SPLINE
SPL {X  -158.227, Y  +353.814, Z    +0.000, E1   +70.663, E3 +51533.806}
SPL {X  -154.257, Y  +335.055, Z    +0.000, E1   +71.089, E3 +51543.434}
SPL {X  -148.153, Y  +317.104, Z    +0.000, E1   +71.658, E3 +51550.580}
SPL {X  -143.479, Y  +306.716, Z    +0.000, E1   +71.847, E3 +51555.654}
SPL {X  -140.298, Y  +300.601, Z    +0.000, E1   +71.461, E3 +51562.409}
SPL {X  -137.001, Y  +294.872, Z    +0.000, E1   +71.048, E3 +51568.917}
SPL {X  -133.301, Y  +289.026, Z    +0.000, E1   +70.567, E3 +51575.704}
SPL {X  -128.648, Y  +282.387, Z    +0.000, E1   +69.939, E3 +51583.519}
SPL {X  -125.063, Y  +277.720, Z    +0.000, E1   +69.378, E3 +51589.095}
SPL {X  -122.086, Y  +274.099, Z    +0.000, E1   +68.932, E3 +51593.340}
SPL {X   -84.117, Y  +241.407, Z    +0.000, E1   +58.224, E3 +51684.223}
ENDSPLINE

SPLINE
SPL {X  -106.708, Y  +258.294, Z    +0.000, E1   +53.789, E3 +51863.010}
SPL {X  -137.973, Y  +296.505, Z    +0.000, E1   +48.844, E3 +51901.790}
SPL {X  -154.359, Y  +335.426, Z    +0.000, E1   +34.338, E3 +51914.686}
SPL {X  -159.279, Y  +362.429, Z    +0.000, E1   +16.013, E3 +51918.286}
SPL {X  -159.976, Y  +375.387, Z    +0.000, E1    +4.229, E3 +51918.937}
SPL {X  -159.990, Y  +379.485, Z    +0.000, E1    +0.028, E3 +51918.982}
SPL {X  -159.990, Y  +381.270, Z    +0.000, E1    -3.383, E3 +51918.999}
SPL {X  -159.990, Y  +384.811, Z    +0.000, E1   -11.531, E3 +51919.089}
SPL {X  -159.990, Y  +390.180, Z    +0.000, E1   -24.142, E3 +51919.392}
SPL {X  -159.990, Y  +397.074, Z    +0.000, E1   -39.012, E3 +51920.002}
SPL {X  -159.990, Y  +405.152, Z    +0.000, E1   -50.697, E3 +51921.141}
SPL {X  -159.990, Y  +423.293, Z    +0.000, E1   -63.280, E3 +51925.143}
SPL {X  -159.990, Y  +493.649, Z    +0.000, E1   -71.671, E3 +51950.847}
SPL {X  -159.990, Y  +662.531, Z    +0.000, E1   -73.010, E3 +52037.670}
SPL {X  -159.805, Y  +684.185, Z    +0.000, E1   -72.979, E3 +52051.954}
SPL {X  -158.739, Y  +696.464, Z    +0.000, E1   -72.862, E3 +52061.072}
SPL {X  -156.417, Y  +710.124, Z    +0.000, E1   -72.650, E3 +52072.296}
SPL {X  -153.206, Y  +722.596, Z    +0.000, E1   -72.287, E3 +52083.734}
SPL {X  -150.445, Y  +730.933, Z    +0.000, E1   -71.979, E3 +52091.944}
SPL {X  -147.389, Y  +738.737, Z    +0.000, E1   -71.634, E3 +52100.017}
SPL {X  -144.044, Y  +746.129, Z    +0.000, E1   -71.236, E3 +52108.011}
SPL {X  -140.684, Y  +752.689, Z    +0.000, E1   -70.820, E3 +52115.387}
SPL {X  -137.335, Y  +758.572, Z    +0.000, E1   -70.388, E3 +52122.194}
SPL {X  -134.566, Y  +763.037, Z    +0.000, E1   -70.007, E3 +52127.490}
SPL {X  -131.456, Y  +767.693, Z    +0.000, E1   -69.587, E3 +52133.054}
SPL {X  -127.440, Y  +773.226, Z    +0.000, E1   -69.006, E3 +52139.737}
SPL {X  -123.127, Y  +778.659, Z    +0.000, E1   -68.349, E3 +52146.279}
SPL {X   -80.879, Y  +814.541, Z    +0.000, E1   -55.704, E3 +52269.184}
ENDSPLINE

SPLINE
SPL {X  -125.518, Y  +775.707, Z    +0.000, E1   -52.189, E3 +52440.661}
SPL {X  -144.748, Y  +744.653, Z    +0.000, E1   -45.208, E3 +52458.857}
SPL {X  -153.147, Y  +722.791, Z    +0.000, E1   -36.417, E3 +52465.252}
SPL {X  -157.402, Y  +705.160, Z    +0.000, E1   -26.108, E3 +52468.348}
SPL {X  -159.480, Y  +689.270, Z    +0.000, E1   -14.023, E3 +52469.913}
SPL {X  -159.986, Y  +677.650, Z    +0.000, E1    -3.291, E3 +52470.408}
SPL {X  -159.990, Y  +674.500, Z    +0.000, E1    +0.000, E3 +52470.438}
SPL {X  -159.990, Y  +672.716, Z    +0.000, E1    +3.405, E3 +52470.455}
SPL {X  -159.990, Y  +668.521, Z    +0.000, E1   +13.007, E3 +52470.574}
SPL {X  -159.990, Y  +662.839, Z    +0.000, E1   +26.519, E3 +52470.916}
SPL {X  -159.990, Y  +653.836, Z    +0.000, E1   +43.967, E3 +52471.846}
SPL {X  -159.990, Y  +641.022, Z    +0.000, E1   +57.726, E3 +52474.155}
SPL {X  -159.990, Y  +617.987, Z    +0.000, E1   +67.134, E3 +52480.051}
SPL {X  -159.990, Y  +532.407, Z    +0.000, E1   +73.084, E3 +52510.957}
SPL {X  -159.990, Y  +382.957, Z    +0.000, E1   +73.647, E3 +52587.217}
SPL {X  -159.615, Y  +366.548, Z    +0.000, E1   +73.602, E3 +52597.859}
SPL {X  -157.928, Y  +351.899, Z    +0.000, E1   +73.451, E3 +52608.714}
ENDSPLINE

SPLINE
SPL {X  -159.990, Y  +380.170, Z    +0.000, E1   +69.785, E3 +52624.854}
ENDSPLINE

SPLINE
SPL {X  -158.227, Y  +353.814, Z    +0.000, E1   +70.663, E3 +52636.748}
SPL {X  -155.560, Y  +340.111, Z    +0.000, E1   +70.976, E3 +52643.770}
SPL {X  -151.918, Y  +327.322, Z    +0.000, E1   +71.266, E3 +52650.113}
SPL {X  -144.697, Y  +309.238, Z    +0.000, E1   +71.848, E3 +52657.063}
SPL {X  -140.298, Y  +300.601, Z    +0.000, E1   +71.461, E3 +52665.350}
SPL {X  -135.903, Y  +293.078, Z    +0.000, E1   +70.930, E3 +52673.888}
SPL {X  -130.487, Y  +284.926, Z    +0.000, E1   +70.202, E3 +52683.447}
SPL {X  -125.807, Y  +278.659, Z    +0.000, E1   +69.508, E3 +52690.904}
SPL {X  -122.967, Y  +275.148, Z    +0.000, E1   +69.053, E3 +52695.073}
SPL {X  -121.236, Y  +273.103, Z    +0.000, E1   +68.779, E3 +52697.458}
SPL {X   -84.117, Y  +241.407, Z    +0.000, E1   +58.224, E3 +52787.164}
ENDSPLINE

SPLINE
SPL {X  -106.708, Y  +258.294, Z    +0.000, E1   +53.789, E3 +52965.951}
SPL {X  -137.973, Y  +296.505, Z    +0.000, E1   +48.844, E3 +53004.731}
SPL {X  -150.692, Y  +323.752, Z    +0.000, E1   +39.895, E3 +53015.097}
SPL {X  -157.053, Y  +346.986, Z    +0.000, E1   +27.437, E3 +53019.577}
SPL {X  -159.518, Y  +365.226, Z    +0.000, E1   +13.562, E3 +53021.442}
SPL {X  -159.976, Y  +375.387, Z    +0.000, E1    +4.229, E3 +53021.878}
SPL {X  -159.990, Y  +379.485, Z    +0.000, E1    +0.028, E3 +53021.923}
SPL {X  -159.990, Y  +381.270, Z    +0.000, E1    -3.383, E3 +53021.940}
SPL {X  -159.990, Y  +384.811, Z    +0.000, E1   -11.531, E3 +53022.030}
SPL {X  -159.990, Y  +390.180, Z    +0.000, E1   -24.142, E3 +53022.333}
SPL {X  -159.990, Y  +397.074, Z    +0.000, E1   -39.012, E3 +53022.943}
SPL {X  -159.990, Y  +405.152, Z    +0.000, E1   -50.697, E3 +53024.082}
SPL {X  -159.990, Y  +423.293, Z    +0.000, E1   -63.280, E3 +53028.084}
SPL {X  -159.990, Y  +493.649, Z    +0.000, E1   -71.671, E3 +53053.788}
SPL {X  -159.990, Y  +662.531, Z    +0.000, E1   -73.010, E3 +53140.611}
SPL {X  -159.805, Y  +684.185, Z    +0.000, E1   -72.979, E3 +53154.895}
SPL {X  -158.739, Y  +696.464, Z    +0.000, E1   -72.862, E3 +53164.014}
SPL {X  -156.417, Y  +710.124, Z    +0.000, E1   -72.650, E3 +53175.237}
SPL {X  -153.206, Y  +722.596, Z    +0.000, E1   -72.287, E3 +53186.675}
SPL {X  -150.445, Y  +730.933, Z    +0.000, E1   -71.979, E3 +53194.885}
SPL {X  -147.389, Y  +738.737, Z    +0.000, E1   -71.634, E3 +53202.958}
SPL {X  -144.044, Y  +746.129, Z    +0.000, E1   -71.236, E3 +53210.952}
SPL {X  -140.684, Y  +752.689, Z    +0.000, E1   -70.820, E3 +53218.328}
SPL {X  -137.335, Y  +758.572, Z    +0.000, E1   -70.388, E3 +53225.135}
SPL {X  -133.651, Y  +764.444, Z    +0.000, E1   -69.897, E3 +53232.087}
SPL {X  -129.492, Y  +770.461, Z    +0.000, E1   -69.311, E3 +53239.327}
SPL {X  -125.168, Y  +776.148, Z    +0.000, E1   -68.666, E3 +53246.204}
SPL {X  -122.036, Y  +779.960, Z    +0.000, E1   -68.144, E3 +53250.807}
SPL {X   -80.879, Y  +814.541, Z    +0.000, E1   -55.704, E3 +53372.125}
ENDSPLINE

SPLINE
SPL {X  -125.518, Y  +775.707, Z    +0.000, E1   -52.189, E3 +53543.602}
SPL {X  -144.748, Y  +744.653, Z    +0.000, E1   -45.208, E3 +53561.798}
SPL {X  -153.147, Y  +722.791, Z    +0.000, E1   -36.417, E3 +53568.194}
SPL {X  -158.456, Y  +698.602, Z    +0.000, E1   -21.523, E3 +53572.040}
SPL {X  -159.738, Y  +685.469, Z    +0.000, E1   -10.595, E3 +53573.094}
SPL {X  -159.986, Y  +677.650, Z    +0.000, E1    -3.291, E3 +53573.349}
SPL {X  -159.990, Y  +674.500, Z    +0.000, E1    +0.000, E3 +53573.379}
SPL {X  -159.990, Y  +672.716, Z    +0.000, E1    +3.405, E3 +53573.396}
SPL {X  -159.990, Y  +668.521, Z    +0.000, E1   +13.007, E3 +53573.515}
SPL {X  -159.990, Y  +662.839, Z    +0.000, E1   +26.519, E3 +53573.857}
SPL {X  -159.990, Y  +653.836, Z    +0.000, E1   +43.967, E3 +53574.787}
SPL {X  -159.990, Y  +641.022, Z    +0.000, E1   +57.726, E3 +53577.096}
SPL {X  -159.990, Y  +617.987, Z    +0.000, E1   +67.134, E3 +53582.992}
SPL {X  -159.990, Y  +532.407, Z    +0.000, E1   +73.084, E3 +53613.899}
SPL {X  -159.990, Y  +382.957, Z    +0.000, E1   +73.647, E3 +53690.158}
SPL {X  -159.615, Y  +366.548, Z    +0.000, E1   +73.602, E3 +53700.801}
SPL {X  -157.928, Y  +351.899, Z    +0.000, E1   +73.451, E3 +53711.655}
ENDSPLINE

SPLINE
SPL {X  -159.990, Y  +380.170, Z    +0.000, E1   +69.785, E3 +53727.795}
ENDSPLINE

SPLINE
SPL {X  -158.227, Y  +353.814, Z    +0.000, E1   +70.663, E3 +53739.689}
SPL {X  -155.560, Y  +340.111, Z    +0.000, E1   +70.976, E3 +53746.711}
SPL {X  -151.918, Y  +327.322, Z    +0.000, E1   +71.266, E3 +53753.054}
SPL {X  -144.697, Y  +309.238, Z    +0.000, E1   +71.848, E3 +53760.004}
SPL {X  -140.298, Y  +300.601, Z    +0.000, E1   +71.461, E3 +53768.292}
SPL {X  -135.903, Y  +293.078, Z    +0.000, E1   +70.930, E3 +53776.829}
SPL {X  -132.382, Y  +287.656, Z    +0.000, E1   +70.425, E3 +53783.221}
SPL {X  -128.648, Y  +282.387, Z    +0.000, E1   +69.939, E3 +53789.402}
SPL {X  -125.063, Y  +277.720, Z    +0.000, E1   +69.378, E3 +53794.977}
SPL {X  -122.086, Y  +274.099, Z    +0.000, E1   +68.932, E3 +53799.223}
SPL {X   -84.117, Y  +241.407, Z    +0.000, E1   +58.224, E3 +53890.105}
ENDSPLINE

SPLINE
SPL {X  -116.986, Y  +268.362, Z    +0.000, E1   +53.233, E3 +54084.021}
SPL {X  -146.319, Y  +312.789, Z    +0.000, E1   +44.152, E3 +54114.487}
SPL {X  -155.980, Y  +341.904, Z    +0.000, E1   +30.583, E3 +54121.782}
SPL {X  -159.279, Y  +362.429, Z    +0.000, E1   +16.013, E3 +54124.168}
SPL {X  -159.976, Y  +375.387, Z    +0.000, E1    +4.229, E3 +54124.819}
SPL {X  -159.990, Y  +379.485, Z    +0.000, E1    +0.028, E3 +54124.864}
SPL {X  -159.990, Y  +381.270, Z    +0.000, E1    -3.383, E3 +54124.881}
SPL {X  -159.990, Y  +386.246, Z    +0.000, E1   -14.704, E3 +54125.039}
SPL {X  -159.990, Y  +394.075, Z    +0.000, E1   -32.836, E3 +54125.599}
SPL {X  -159.990, Y  +405.152, Z    +0.000, E1   -50.697, E3 +54127.024}
SPL {X  -159.990, Y  +423.293, Z    +0.000, E1   -63.280, E3 +54131.025}
SPL {X  -159.990, Y  +493.649, Z    +0.000, E1   -71.671, E3 +54156.729}
SPL {X  -159.990, Y  +662.531, Z    +0.000, E1   -73.010, E3 +54243.552}
SPL {X  -159.805, Y  +684.185, Z    +0.000, E1   -72.979, E3 +54257.836}
SPL {X  -158.295, Y  +699.729, Z    +0.000, E1   -72.830, E3 +54269.506}
SPL {X  -155.857, Y  +712.630, Z    +0.000, E1   -72.572, E3 +54280.435}
SPL {X  -153.206, Y  +722.596, Z    +0.000, E1   -72.287, E3 +54289.616}
SPL {X  -150.445, Y  +730.933, Z    +0.000, E1   -71.979, E3 +54297.827}
SPL {X  -147.389, Y  +738.737, Z    +0.000, E1   -71.634, E3 +54305.899}
SPL {X  -144.044, Y  +746.129, Z    +0.000, E1   -71.236, E3 +54313.894}
SPL {X  -140.684, Y  +752.689, Z    +0.000, E1   -70.820, E3 +54321.269}
SPL {X  -137.335, Y  +758.572, Z    +0.000, E1   -70.388, E3 +54328.076}
SPL {X  -133.651, Y  +764.444, Z    +0.000, E1   -69.897, E3 +54335.028}
SPL {X  -129.492, Y  +770.461, Z    +0.000, E1   -69.311, E3 +54342.269}
SPL {X  -125.168, Y  +776.148, Z    +0.000, E1   -68.666, E3 +54349.145}
SPL {X  -122.036, Y  +779.960, Z    +0.000, E1   -68.144, E3 +54353.748}
SPL {X   -80.879, Y  +814.541, Z    +0.000, E1   -55.704, E3 +54475.066}
ENDSPLINE

SPLINE
SPL {X  -125.518, Y  +775.707, Z    +0.000, E1   -52.189, E3 +54646.543}
SPL {X  -144.748, Y  +744.653, Z    +0.000, E1   -45.208, E3 +54664.739}
SPL {X  -153.147, Y  +722.791, Z    +0.000, E1   -36.417, E3 +54671.135}
SPL {X  -157.402, Y  +705.160, Z    +0.000, E1   -26.108, E3 +54674.230}
SPL {X  -159.480, Y  +689.270, Z    +0.000, E1   -14.023, E3 +54675.796}
SPL {X  -159.986, Y  +677.650, Z    +0.000, E1    -3.291, E3 +54676.290}
SPL {X  -159.990, Y  +674.500, Z    +0.000, E1    +0.000, E3 +54676.320}
SPL {X  -159.990, Y  +672.716, Z    +0.000, E1    +3.405, E3 +54676.337}
SPL {X  -159.990, Y  +668.521, Z    +0.000, E1   +13.007, E3 +54676.456}
SPL {X  -159.990, Y  +664.286, Z    +0.000, E1   +23.338, E3 +54676.688}
SPL {X  -159.990, Y  +658.431, Z    +0.000, E1   +35.998, E3 +54677.182}
SPL {X  -159.990, Y  +650.524, Z    +0.000, E1   +48.779, E3 +54678.171}
SPL {X  -159.990, Y  +641.022, Z    +0.000, E1   +57.726, E3 +54680.038}
SPL {X  -159.990, Y  +617.987, Z    +0.000, E1   +67.134, E3 +54685.933}
SPL {X  -159.990, Y  +532.407, Z    +0.000, E1   +73.084, E3 +54716.840}
SPL {X  -159.990, Y  +390.607, Z    +0.000, E1   +73.632, E3 +54788.376}
SPL {X  -159.886, Y  +371.742, Z    +0.000, E1   +73.650, E3 +54800.163}
SPL {X  -157.928, Y  +351.899, Z    +0.000, E1   +73.451, E3 +54814.596}
ENDSPLINE

SPLINE
SPL {X  -159.990, Y  +380.170, Z    +0.000, E1   +69.785, E3 +54830.736}
ENDSPLINE

SPLINE
SPL {X  -158.227, Y  +353.814, Z    +0.000, E1   +70.663, E3 +54842.630}
SPL {X  -154.257, Y  +335.055, Z    +0.000, E1   +71.089, E3 +54852.258}
SPL {X  -148.153, Y  +317.104, Z    +0.000, E1   +71.658, E3 +54859.404}
SPL {X  -143.479, Y  +306.716, Z    +0.000, E1   +71.847, E3 +54864.477}
SPL {X  -140.298, Y  +300.601, Z    +0.000, E1   +71.461, E3 +54871.233}
SPL {X  -137.001, Y  +294.872, Z    +0.000, E1   +71.048, E3 +54877.741}
SPL {X  -133.301, Y  +289.026, Z    +0.000, E1   +70.567, E3 +54884.527}
SPL {X  -129.603, Y  +283.692, Z    +0.000, E1   +70.051, E3 +54890.827}
SPL {X  -125.807, Y  +278.659, Z    +0.000, E1   +69.508, E3 +54896.786}
SPL {X  -122.086, Y  +274.099, Z    +0.000, E1   +68.932, E3 +54902.164}
SPL {X   -84.117, Y  +241.407, Z    +0.000, E1   +58.224, E3 +54993.046}
ENDSPLINE

SPLINE
SPL {X  -116.986, Y  +268.362, Z    +0.000, E1   +53.233, E3 +55186.962}
SPL {X  -146.319, Y  +312.789, Z    +0.000, E1   +44.152, E3 +55217.428}
SPL {X  -157.053, Y  +346.986, Z    +0.000, E1   +27.437, E3 +55225.459}
SPL {X  -159.518, Y  +365.226, Z    +0.000, E1   +13.562, E3 +55227.325}
SPL {X  -159.976, Y  +375.387, Z    +0.000, E1    +4.229, E3 +55227.760}
SPL {X  -159.990, Y  +379.485, Z    +0.000, E1    +0.028, E3 +55227.805}
SPL {X  -159.990, Y  +381.270, Z    +0.000, E1    -3.383, E3 +55227.822}
SPL {X  -159.990, Y  +386.246, Z    +0.000, E1   -14.704, E3 +55227.980}
SPL {X  -159.990, Y  +394.075, Z    +0.000, E1   -32.836, E3 +55228.541}
SPL {X  -159.990, Y  +405.152, Z    +0.000, E1   -50.697, E3 +55229.965}
SPL {X  -159.990, Y  +423.293, Z    +0.000, E1   -63.280, E3 +55233.966}
SPL {X  -159.990, Y  +493.649, Z    +0.000, E1   -71.671, E3 +55259.670}
SPL {X  -159.990, Y  +662.531, Z    +0.000, E1   -73.010, E3 +55346.493}
SPL {X  -159.805, Y  +684.185, Z    +0.000, E1   -72.979, E3 +55360.777}
SPL {X  -158.295, Y  +699.729, Z    +0.000, E1   -72.830, E3 +55372.447}
SPL {X  -155.857, Y  +712.630, Z    +0.000, E1   -72.572, E3 +55383.376}
SPL {X  -153.206, Y  +722.596, Z    +0.000, E1   -72.287, E3 +55392.557}
SPL {X  -150.445, Y  +730.933, Z    +0.000, E1   -71.979, E3 +55400.768}
SPL {X  -147.389, Y  +738.737, Z    +0.000, E1   -71.634, E3 +55408.840}
SPL {X  -144.044, Y  +746.129, Z    +0.000, E1   -71.236, E3 +55416.835}
SPL {X  -140.684, Y  +752.689, Z    +0.000, E1   -70.820, E3 +55424.210}
SPL {X  -136.099, Y  +760.606, Z    +0.000, E1   -70.253, E3 +55433.366}
SPL {X  -131.456, Y  +767.693, Z    +0.000, E1   -69.587, E3 +55441.877}
SPL {X  -127.440, Y  +773.226, Z    +0.000, E1   -69.006, E3 +55448.561}
SPL {X  -123.127, Y  +778.659, Z    +0.000, E1   -68.349, E3 +55455.103}
SPL {X   -80.879, Y  +814.541, Z    +0.000, E1   -55.704, E3 +55578.007}
ENDSPLINE

SPLINE
SPL {X  -125.518, Y  +775.707, Z    +0.000, E1   -52.189, E3 +55749.484}
SPL {X  -150.797, Y  +729.951, Z    +0.000, E1   -39.777, E3 +55772.219}
SPL {X  -157.402, Y  +705.160, Z    +0.000, E1   -26.108, E3 +55777.171}
SPL {X  -159.480, Y  +689.270, Z    +0.000, E1   -14.023, E3 +55778.737}
SPL {X  -159.986, Y  +677.650, Z    +0.000, E1    -3.291, E3 +55779.231}
SPL {X  -159.990, Y  +674.500, Z    +0.000, E1    +0.000, E3 +55779.262}
SPL {X  -159.990, Y  +672.716, Z    +0.000, E1    +3.405, E3 +55779.278}
SPL {X  -159.990, Y  +668.521, Z    +0.000, E1   +13.007, E3 +55779.397}
SPL {X  -159.990, Y  +662.839, Z    +0.000, E1   +26.519, E3 +55779.740}
SPL {X  -159.990, Y  +653.836, Z    +0.000, E1   +43.967, E3 +55780.670}
SPL {X  -159.990, Y  +641.022, Z    +0.000, E1   +57.726, E3 +55782.979}
SPL {X  -159.990, Y  +617.987, Z    +0.000, E1   +67.134, E3 +55788.874}
SPL {X  -159.990, Y  +532.407, Z    +0.000, E1   +73.084, E3 +55819.781}
SPL {X  -159.990, Y  +390.607, Z    +0.000, E1   +73.632, E3 +55891.317}
SPL {X  -159.886, Y  +371.742, Z    +0.000, E1   +73.650, E3 +55903.104}
SPL {X  -157.928, Y  +351.899, Z    +0.000, E1   +73.451, E3 +55917.537}
ENDSPLINE

SPLINE
SPL {X  -159.990, Y  +380.170, Z    +0.000, E1   +69.785, E3 +55933.678}
ENDSPLINE

SPLINE
SPL {X  -158.227, Y  +353.814, Z    +0.000, E1   +70.663, E3 +55945.571}
SPL {X  -155.560, Y  +340.111, Z    +0.000, E1   +70.976, E3 +55952.593}
SPL {X  -151.918, Y  +327.322, Z    +0.000, E1   +71.266, E3 +55958.937}
SPL {X  -144.697, Y  +309.238, Z    +0.000, E1   +71.848, E3 +55965.886}
SPL {X  -140.298, Y  +300.601, Z    +0.000, E1   +71.461, E3 +55974.174}
SPL {X  -135.903, Y  +293.078, Z    +0.000, E1   +70.930, E3 +55982.712}
SPL {X  -130.487, Y  +284.926, Z    +0.000, E1   +70.202, E3 +55992.271}
SPL {X  -125.807, Y  +278.659, Z    +0.000, E1   +69.508, E3 +55999.727}
SPL {X  -122.967, Y  +275.148, Z    +0.000, E1   +69.053, E3 +56003.896}
SPL {X  -121.236, Y  +273.103, Z    +0.000, E1   +68.779, E3 +56006.282}
SPL {X   -84.117, Y  +241.407, Z    +0.000, E1   +58.224, E3 +56095.988}
ENDSPLINE

SPLINE
SPL {X  -116.986, Y  +268.362, Z    +0.000, E1   +53.233, E3 +56289.903}
SPL {X  -146.319, Y  +312.789, Z    +0.000, E1   +44.152, E3 +56320.369}
SPL {X  -157.053, Y  +346.986, Z    +0.000, E1   +27.437, E3 +56328.400}
SPL {X  -159.518, Y  +365.226, Z    +0.000, E1   +13.562, E3 +56330.266}
SPL {X  -159.976, Y  +375.387, Z    +0.000, E1    +4.229, E3 +56330.701}
SPL {X  -159.990, Y  +379.485, Z    +0.000, E1    +0.028, E3 +56330.746}
SPL {X  -159.990, Y  +381.270, Z    +0.000, E1    -3.383, E3 +56330.764}
SPL {X  -159.990, Y  +386.246, Z    +0.000, E1   -14.704, E3 +56330.921}
SPL {X  -159.990, Y  +394.075, Z    +0.000, E1   -32.836, E3 +56331.482}
SPL {X  -159.990, Y  +405.152, Z    +0.000, E1   -50.697, E3 +56332.906}
SPL {X  -159.990, Y  +423.293, Z    +0.000, E1   -63.280, E3 +56336.907}
SPL {X  -159.990, Y  +493.649, Z    +0.000, E1   -71.671, E3 +56362.611}
SPL {X  -159.990, Y  +662.531, Z    +0.000, E1   -73.010, E3 +56449.434}
SPL {X  -159.805, Y  +684.185, Z    +0.000, E1   -72.979, E3 +56463.718}
SPL {X  -158.295, Y  +699.729, Z    +0.000, E1   -72.830, E3 +56475.389}
SPL {X  -155.857, Y  +712.630, Z    +0.000, E1   -72.572, E3 +56486.318}
SPL {X  -153.206, Y  +722.596, Z    +0.000, E1   -72.287, E3 +56495.499}
SPL {X  -150.445, Y  +730.933, Z    +0.000, E1   -71.979, E3 +56503.709}
SPL {X  -147.389, Y  +738.737, Z    +0.000, E1   -71.634, E3 +56511.782}
SPL {X  -144.044, Y  +746.129, Z    +0.000, E1   -71.236, E3 +56519.776}
SPL {X  -140.684, Y  +752.689, Z    +0.000, E1   -70.820, E3 +56527.151}
SPL {X  -136.099, Y  +760.606, Z    +0.000, E1   -70.253, E3 +56536.307}
SPL {X  -131.456, Y  +767.693, Z    +0.000, E1   -69.587, E3 +56544.818}
SPL {X  -127.440, Y  +773.226, Z    +0.000, E1   -69.006, E3 +56551.502}
SPL {X  -123.127, Y  +778.659, Z    +0.000, E1   -68.349, E3 +56558.044}
SPL {X   -80.879, Y  +814.541, Z    +0.000, E1   -55.704, E3 +56680.948}
ENDSPLINE

SPLINE
SPL {X  -125.518, Y  +775.707, Z    +0.000, E1   -52.189, E3 +56852.426}
SPL {X  -150.797, Y  +729.951, Z    +0.000, E1   -39.777, E3 +56875.161}
SPL {X  -158.456, Y  +698.602, Z    +0.000, E1   -21.523, E3 +56880.863}
SPL {X  -159.738, Y  +685.469, Z    +0.000, E1   -10.595, E3 +56881.918}
SPL {X  -159.986, Y  +677.650, Z    +0.000, E1    -3.291, E3 +56882.172}
SPL {X  -159.990, Y  +674.500, Z    +0.000, E1    +0.000, E3 +56882.203}
SPL {X  -159.990, Y  +672.716, Z    +0.000, E1    +3.405, E3 +56882.219}
SPL {X  -159.990, Y  +668.521, Z    +0.000, E1   +13.007, E3 +56882.338}
SPL {X  -159.990, Y  +662.839, Z    +0.000, E1   +26.519, E3 +56882.681}
SPL {X  -159.990, Y  +653.836, Z    +0.000, E1   +43.967, E3 +56883.611}
SPL {X  -159.990, Y  +641.022, Z    +0.000, E1   +57.726, E3 +56885.920}
SPL {X  -159.990, Y  +617.987, Z    +0.000, E1   +67.134, E3 +56891.815}
SPL {X  -159.990, Y  +532.407, Z    +0.000, E1   +73.084, E3 +56922.722}
SPL {X  -159.990, Y  +382.957, Z    +0.000, E1   +73.647, E3 +56998.982}
SPL {X  -159.615, Y  +366.548, Z    +0.000, E1   +73.602, E3 +57009.624}
SPL {X  -157.928, Y  +351.899, Z    +0.000, E1   +73.451, E3 +57020.479}
ENDSPLINE

SPLINE
SPL {X  -159.990, Y  +380.170, Z    +0.000, E1   +69.785, E3 +57036.619}
ENDSPLINE

SPLINE
SPL {X  -158.227, Y  +353.814, Z    +0.000, E1   +70.663, E3 +57048.512}
SPL {X  -154.257, Y  +335.055, Z    +0.000, E1   +71.089, E3 +57058.140}
SPL {X  -148.153, Y  +317.104, Z    +0.000, E1   +71.658, E3 +57065.286}
SPL {X  -143.479, Y  +306.716, Z    +0.000, E1   +71.847, E3 +57070.359}
SPL {X  -140.298, Y  +300.601, Z    +0.000, E1   +71.461, E3 +57077.115}
SPL {X  -137.001, Y  +294.872, Z    +0.000, E1   +71.048, E3 +57083.623}
SPL {X  -133.301, Y  +289.026, Z    +0.000, E1   +70.567, E3 +57090.410}
SPL {X  -128.648, Y  +282.387, Z    +0.000, E1   +69.939, E3 +57098.225}
SPL {X  -125.063, Y  +277.720, Z    +0.000, E1   +69.378, E3 +57103.801}
SPL {X  -122.086, Y  +274.099, Z    +0.000, E1   +68.932, E3 +57108.046}
SPL {X   -84.117, Y  +241.407, Z    +0.000, E1   +58.224, E3 +57198.929}
ENDSPLINE

SPLINE
SPL {X  -106.708, Y  +258.294, Z    +0.000, E1   +53.789, E3 +57377.716}
SPL {X  -137.973, Y  +296.505, Z    +0.000, E1   +48.844, E3 +57416.496}
SPL {X  -154.359, Y  +335.426, Z    +0.000, E1   +34.338, E3 +57429.392}
SPL {X  -159.279, Y  +362.429, Z    +0.000, E1   +16.013, E3 +57432.992}
SPL {X  -159.976, Y  +375.387, Z    +0.000, E1    +4.229, E3 +57433.643}
SPL {X  -159.990, Y  +379.485, Z    +0.000, E1    +0.028, E3 +57433.688}
SPL {X  -159.990, Y  +381.270, Z    +0.000, E1    -3.383, E3 +57433.705}
SPL {X  -159.990, Y  +386.246, Z    +0.000, E1   -14.704, E3 +57433.862}
SPL {X  -159.990, Y  +394.075, Z    +0.000, E1   -32.836, E3 +57434.423}
SPL {X  -159.990, Y  +405.152, Z    +0.000, E1   -50.697, E3 +57435.847}
SPL {X  -159.990, Y  +423.293, Z    +0.000, E1   -63.280, E3 +57439.849}
SPL {X  -159.990, Y  +493.649, Z    +0.000, E1   -71.671, E3 +57465.552}
SPL {X  -159.990, Y  +662.531, Z    +0.000, E1   -73.010, E3 +57552.376}
SPL {X  -159.805, Y  +684.185, Z    +0.000, E1   -72.979, E3 +57566.660}
SPL {X  -158.739, Y  +696.464, Z    +0.000, E1   -72.862, E3 +57575.778}
SPL {X  -156.417, Y  +710.124, Z    +0.000, E1   -72.650, E3 +57587.002}
SPL {X  -153.206, Y  +722.596, Z    +0.000, E1   -72.287, E3 +57598.440}
SPL {X  -150.445, Y  +730.933, Z    +0.000, E1   -71.979, E3 +57606.650}
SPL {X  -147.389, Y  +738.737, Z    +0.000, E1   -71.634, E3 +57614.723}
SPL {X  -144.044, Y  +746.129, Z    +0.000, E1   -71.236, E3 +57622.717}
SPL {X  -140.684, Y  +752.689, Z    +0.000, E1   -70.820, E3 +57630.092}
SPL {X  -136.099, Y  +760.606, Z    +0.000, E1   -70.253, E3 +57639.248}
SPL {X  -131.456, Y  +767.693, Z    +0.000, E1   -69.587, E3 +57647.760}
SPL {X  -127.440, Y  +773.226, Z    +0.000, E1   -69.006, E3 +57654.443}
SPL {X  -123.127, Y  +778.659, Z    +0.000, E1   -68.349, E3 +57660.985}
SPL {X   -80.879, Y  +814.541, Z    +0.000, E1   -55.704, E3 +57783.889}
ENDSPLINE

SPLINE
SPL {X  -125.518, Y  +775.707, Z    +0.000, E1   -52.189, E3 +57955.367}
SPL {X  -144.748, Y  +744.653, Z    +0.000, E1   -45.208, E3 +57973.563}
SPL {X  -153.147, Y  +722.791, Z    +0.000, E1   -36.417, E3 +57979.958}
SPL {X  -158.456, Y  +698.602, Z    +0.000, E1   -21.523, E3 +57983.804}
SPL {X  -159.738, Y  +685.469, Z    +0.000, E1   -10.595, E3 +57984.859}
SPL {X  -159.986, Y  +677.650, Z    +0.000, E1    -3.291, E3 +57985.114}
SPL {X  -159.990, Y  +674.500, Z    +0.000, E1    +0.000, E3 +57985.144}
SPL {X  -159.990, Y  +672.716, Z    +0.000, E1    +3.405, E3 +57985.161}
SPL {X  -159.990, Y  +668.521, Z    +0.000, E1   +13.007, E3 +57985.280}
SPL {X  -159.990, Y  +662.839, Z    +0.000, E1   +26.519, E3 +57985.622}
SPL {X  -159.990, Y  +653.836, Z    +0.000, E1   +43.967, E3 +57986.552}
SPL {X  -159.990, Y  +641.022, Z    +0.000, E1   +57.726, E3 +57988.861}
SPL {X  -159.990, Y  +617.987, Z    +0.000, E1   +67.134, E3 +57994.757}
SPL {X  -159.990, Y  +532.407, Z    +0.000, E1   +73.084, E3 +58025.663}
SPL {X  -159.990, Y  +390.607, Z    +0.000, E1   +73.632, E3 +58097.199}
SPL {X  -159.886, Y  +371.742, Z    +0.000, E1   +73.650, E3 +58108.986}
SPL {X  -157.928, Y  +351.899, Z    +0.000, E1   +73.451, E3 +58123.420}
ENDSPLINE

SPLINE
SPL {X  -159.990, Y  +387.996, Z    +0.000, E1   +69.509, E3 +58135.850}
ENDSPLINE

SPLINE
SPL {X  -159.889, Y  +371.819, Z    +0.000, E1   +70.046, E3 +58143.577}
SPL {X  -158.227, Y  +353.814, Z    +0.000, E1   +70.663, E3 +58151.454}
SPL {X  -154.257, Y  +335.055, Z    +0.000, E1   +71.089, E3 +58161.082}
SPL {X  -148.153, Y  +317.104, Z    +0.000, E1   +71.658, E3 +58168.227}
SPL {X  -143.479, Y  +306.716, Z    +0.000, E1   +71.847, E3 +58173.301}
SPL {X  -140.298, Y  +300.601, Z    +0.000, E1   +71.461, E3 +58180.056}
SPL {X  -135.903, Y  +293.078, Z    +0.000, E1   +70.930, E3 +58188.594}
SPL {X  -130.487, Y  +284.926, Z    +0.000, E1   +70.202, E3 +58198.153}
SPL {X  -125.807, Y  +278.659, Z    +0.000, E1   +69.508, E3 +58205.610}
SPL {X  -122.967, Y  +275.148, Z    +0.000, E1   +69.053, E3 +58209.779}
SPL {X  -121.236, Y  +273.103, Z    +0.000, E1   +68.779, E3 +58212.164}
SPL {X   -84.117, Y  +241.407, Z    +0.000, E1   +58.224, E3 +58301.870}
ENDSPLINE

SPLINE
SPL {X  -116.986, Y  +268.362, Z    +0.000, E1   +53.233, E3 +58495.785}
SPL {X  -146.319, Y  +312.789, Z    +0.000, E1   +44.152, E3 +58526.252}
SPL {X  -157.053, Y  +346.986, Z    +0.000, E1   +27.437, E3 +58534.283}
SPL {X  -159.518, Y  +365.226, Z    +0.000, E1   +13.562, E3 +58536.148}
SPL {X  -159.976, Y  +375.387, Z    +0.000, E1    +4.229, E3 +58536.584}
SPL {X  -159.990, Y  +379.485, Z    +0.000, E1    +0.028, E3 +58536.629}
SPL {X  -159.990, Y  +381.270, Z    +0.000, E1    -3.383, E3 +58536.646}
SPL {X  -159.990, Y  +384.811, Z    +0.000, E1   -11.531, E3 +58536.736}
SPL {X  -159.990, Y  +388.002, Z    +0.000, E1   -19.281, E3 +58536.886}
SPL {X  -159.990, Y  +394.075, Z    +0.000, E1   -32.836, E3 +58537.364}
SPL {X  -159.990, Y  +405.152, Z    +0.000, E1   -50.697, E3 +58538.788}
SPL {X  -159.990, Y  +423.293, Z    +0.000, E1   -63.280, E3 +58542.790}
SPL {X  -159.990, Y  +493.649, Z    +0.000, E1   -71.671, E3 +58568.494}
SPL {X  -159.990, Y  +654.929, Z    +0.000, E1   -72.988, E3 +58650.443}
SPL {X  -159.990, Y  +668.018, Z    +0.000, E1   -72.989, E3 +58658.936}
SPL {X  -159.805, Y  +684.185, Z    +0.000, E1   -72.979, E3 +58669.601}
SPL {X  -158.295, Y  +699.729, Z    +0.000, E1   -72.830, E3 +58681.271}
SPL {X  -155.857, Y  +712.630, Z    +0.000, E1   -72.572, E3 +58692.200}
SPL {X  -153.206, Y  +722.596, Z    +0.000, E1   -72.287, E3 +58701.381}
SPL {X  -150.445, Y  +730.933, Z    +0.000, E1   -71.979, E3 +58709.591}
SPL {X  -147.389, Y  +738.737, Z    +0.000, E1   -71.634, E3 +58717.664}
SPL {X  -144.044, Y  +746.129, Z    +0.000, E1   -71.236, E3 +58725.658}
SPL {X  -140.684, Y  +752.689, Z    +0.000, E1   -70.820, E3 +58733.034}
SPL {X  -136.099, Y  +760.606, Z    +0.000, E1   -70.253, E3 +58742.189}
SPL {X  -131.456, Y  +767.693, Z    +0.000, E1   -69.587, E3 +58750.701}
SPL {X  -128.507, Y  +771.803, Z    +0.000, E1   -69.145, E3 +58755.683}
SPL {X  -125.168, Y  +776.148, Z    +0.000, E1   -68.666, E3 +58760.910}
SPL {X  -122.036, Y  +779.960, Z    +0.000, E1   -68.144, E3 +58765.513}
SPL {X   -80.879, Y  +814.541, Z    +0.000, E1   -55.704, E3 +58886.831}
ENDSPLINE

SPLINE
SPL {X  -125.518, Y  +775.707, Z    +0.000, E1   -52.189, E3 +59058.308}
SPL {X  -144.748, Y  +744.653, Z    +0.000, E1   -45.208, E3 +59076.504}
SPL {X  -153.147, Y  +722.791, Z    +0.000, E1   -36.417, E3 +59082.900}
SPL {X  -158.456, Y  +698.602, Z    +0.000, E1   -21.523, E3 +59086.746}
SPL {X  -159.738, Y  +685.469, Z    +0.000, E1   -10.595, E3 +59087.800}
SPL {X  -159.986, Y  +677.650, Z    +0.000, E1    -3.291, E3 +59088.055}
SPL {X  -159.990, Y  +674.500, Z    +0.000, E1    +0.000, E3 +59088.085}
SPL {X  -159.990, Y  +672.716, Z    +0.000, E1    +3.405, E3 +59088.102}
SPL {X  -159.990, Y  +668.521, Z    +0.000, E1   +13.007, E3 +59088.221}
SPL {X  -159.990, Y  +664.286, Z    +0.000, E1   +23.338, E3 +59088.452}
SPL {X  -159.990, Y  +658.431, Z    +0.000, E1   +35.998, E3 +59088.947}
SPL {X  -159.990, Y  +650.524, Z    +0.000, E1   +48.779, E3 +59089.935}
SPL {X  -159.990, Y  +641.022, Z    +0.000, E1   +57.726, E3 +59091.802}
SPL {X  -159.990, Y  +617.987, Z    +0.000, E1   +67.134, E3 +59097.698}
SPL {X  -159.990, Y  +532.407, Z    +0.000, E1   +73.084, E3 +59128.605}
SPL {X  -159.990, Y  +382.957, Z    +0.000, E1   +73.647, E3 +59204.864}
SPL {X  -159.615, Y  +366.548, Z    +0.000, E1   +73.602, E3 +59215.507}
SPL {X  -157.928, Y  +351.899, Z    +0.000, E1   +73.451, E3 +59226.361}
ENDSPLINE

SPLINE
SPL {X  -159.990, Y  +380.170, Z    +0.000, E1   +69.785, E3 +59242.501}
ENDSPLINE

SPLINE
SPL {X  -158.227, Y  +353.814, Z    +0.000, E1   +70.663, E3 +59254.395}
SPL {X  -155.560, Y  +340.111, Z    +0.000, E1   +70.976, E3 +59261.417}
SPL {X  -151.918, Y  +327.322, Z    +0.000, E1   +71.266, E3 +59267.760}
SPL {X  -144.697, Y  +309.238, Z    +0.000, E1   +71.848, E3 +59274.710}
SPL {X  -140.298, Y  +300.601, Z    +0.000, E1   +71.461, E3 +59282.997}
SPL {X  -137.001, Y  +294.872, Z    +0.000, E1   +71.048, E3 +59289.506}
SPL {X  -133.301, Y  +289.026, Z    +0.000, E1   +70.567, E3 +59296.292}
SPL {X  -128.648, Y  +282.387, Z    +0.000, E1   +69.939, E3 +59304.107}
SPL {X  -125.063, Y  +277.720, Z    +0.000, E1   +69.378, E3 +59309.683}
SPL {X  -122.086, Y  +274.099, Z    +0.000, E1   +68.932, E3 +59313.928}
SPL {X   -84.117, Y  +241.407, Z    +0.000, E1   +58.224, E3 +59404.811}
ENDSPLINE

SPLINE
SPL {X  -106.708, Y  +258.294, Z    +0.000, E1   +53.789, E3 +59583.598}
SPL {X  -137.973, Y  +296.505, Z    +0.000, E1   +48.844, E3 +59622.378}
SPL {X  -154.359, Y  +335.426, Z    +0.000, E1   +34.338, E3 +59635.274}
SPL {X  -159.279, Y  +362.429, Z    +0.000, E1   +16.013, E3 +59638.874}
SPL {X  -159.976, Y  +375.387, Z    +0.000, E1    +4.229, E3 +59639.525}
SPL {X  -159.990, Y  +379.485, Z    +0.000, E1    +0.028, E3 +59639.570}
SPL {X  -159.990, Y  +381.270, Z    +0.000, E1    -3.383, E3 +59639.587}
SPL {X  -159.990, Y  +384.811, Z    +0.000, E1   -11.531, E3 +59639.677}
SPL {X  -159.990, Y  +390.180, Z    +0.000, E1   -24.142, E3 +59639.980}
SPL {X  -159.990, Y  +397.074, Z    +0.000, E1   -39.012, E3 +59640.590}
SPL {X  -159.990, Y  +405.152, Z    +0.000, E1   -50.697, E3 +59641.730}
SPL {X  -159.990, Y  +423.293, Z    +0.000, E1   -63.280, E3 +59645.731}
SPL {X  -159.990, Y  +493.649, Z    +0.000, E1   -71.671, E3 +59671.435}
SPL {X  -159.990, Y  +662.531, Z    +0.000, E1   -73.010, E3 +59758.258}
SPL {X  -159.805, Y  +684.185, Z    +0.000, E1   -72.979, E3 +59772.542}
SPL {X  -158.295, Y  +699.729, Z    +0.000, E1   -72.830, E3 +59784.212}
SPL {X  -155.857, Y  +712.630, Z    +0.000, E1   -72.572, E3 +59795.141}
SPL {X  -153.206, Y  +722.596, Z    +0.000, E1   -72.287, E3 +59804.322}
SPL {X  -150.445, Y  +730.933, Z    +0.000, E1   -71.979, E3 +59812.532}
SPL {X  -147.389, Y  +738.737, Z    +0.000, E1   -71.634, E3 +59820.605}
SPL {X  -144.044, Y  +746.129, Z    +0.000, E1   -71.236, E3 +59828.600}
SPL {X  -140.684, Y  +752.689, Z    +0.000, E1   -70.820, E3 +59835.975}
SPL {X  -137.335, Y  +758.572, Z    +0.000, E1   -70.388, E3 +59842.782}
SPL {X  -133.651, Y  +764.444, Z    +0.000, E1   -69.897, E3 +59849.734}
SPL {X  -129.492, Y  +770.461, Z    +0.000, E1   -69.311, E3 +59856.974}
SPL {X  -125.168, Y  +776.148, Z    +0.000, E1   -68.666, E3 +59863.851}
SPL {X  -122.036, Y  +779.960, Z    +0.000, E1   -68.144, E3 +59868.454}
SPL {X   -80.879, Y  +814.541, Z    +0.000, E1   -55.704, E3 +59989.772}
ENDSPLINE

SPLINE
SPL {X  -125.518, Y  +775.707, Z    +0.000, E1   -52.189, E3 +60161.249}
SPL {X  -144.748, Y  +744.653, Z    +0.000, E1   -45.208, E3 +60179.445}
SPL {X  -153.147, Y  +722.791, Z    +0.000, E1   -36.417, E3 +60185.841}
SPL {X  -157.402, Y  +705.160, Z    +0.000, E1   -26.108, E3 +60188.936}
SPL {X  -159.480, Y  +689.270, Z    +0.000, E1   -14.023, E3 +60190.502}
SPL {X  -159.986, Y  +677.650, Z    +0.000, E1    -3.291, E3 +60190.996}
SPL {X  -159.990, Y  +674.500, Z    +0.000, E1    +0.000, E3 +60191.026}
SPL {X  -159.990, Y  +672.716, Z    +0.000, E1    +3.405, E3 +60191.043}
SPL {X  -159.990, Y  +668.521, Z    +0.000, E1   +13.007, E3 +60191.162}
SPL {X  -159.990, Y  +664.286, Z    +0.000, E1   +23.338, E3 +60191.393}
SPL {X  -159.990, Y  +658.431, Z    +0.000, E1   +35.998, E3 +60191.888}
SPL {X  -159.990, Y  +650.524, Z    +0.000, E1   +48.779, E3 +60192.877}
SPL {X  -159.990, Y  +641.022, Z    +0.000, E1   +57.726, E3 +60194.743}
SPL {X  -159.990, Y  +617.987, Z    +0.000, E1   +67.134, E3 +60200.639}
SPL {X  -159.990, Y  +532.407, Z    +0.000, E1   +73.084, E3 +60231.546}
SPL {X  -159.990, Y  +390.607, Z    +0.000, E1   +73.632, E3 +60303.082}
SPL {X  -159.886, Y  +371.742, Z    +0.000, E1   +73.650, E3 +60314.869}
SPL {X  -157.928, Y  +351.899, Z    +0.000, E1   +73.451, E3 +60329.302}
ENDSPLINE

SPLINE
SPL {X  -159.990, Y  +380.170, Z    +0.000, E1   +69.785, E3 +60345.442}
ENDSPLINE

SPLINE
SPL {X  -158.227, Y  +353.814, Z    +0.000, E1   +70.663, E3 +60357.336}
SPL {X  -155.560, Y  +340.111, Z    +0.000, E1   +70.976, E3 +60364.358}
SPL {X  -151.918, Y  +327.322, Z    +0.000, E1   +71.266, E3 +60370.702}
SPL {X  -144.697, Y  +309.238, Z    +0.000, E1   +71.848, E3 +60377.651}
SPL {X  -140.298, Y  +300.601, Z    +0.000, E1   +71.461, E3 +60385.939}
SPL {X  -137.001, Y  +294.872, Z    +0.000, E1   +71.048, E3 +60392.447}
SPL {X  -133.301, Y  +289.026, Z    +0.000, E1   +70.567, E3 +60399.233}
SPL {X  -129.603, Y  +283.692, Z    +0.000, E1   +70.051, E3 +60405.533}
SPL {X  -125.807, Y  +278.659, Z    +0.000, E1   +69.508, E3 +60411.492}
SPL {X  -122.086, Y  +274.099, Z    +0.000, E1   +68.932, E3 +60416.870}
SPL {X   -84.117, Y  +241.407, Z    +0.000, E1   +58.224, E3 +60507.752}
ENDSPLINE

SPLINE
SPL {X  -106.708, Y  +258.294, Z    +0.000, E1   +53.789, E3 +60686.539}
SPL {X  -137.973, Y  +296.505, Z    +0.000, E1   +48.844, E3 +60725.319}
SPL {X  -154.359, Y  +335.426, Z    +0.000, E1   +34.338, E3 +60738.215}
SPL {X  -159.279, Y  +362.429, Z    +0.000, E1   +16.013, E3 +60741.815}
SPL {X  -159.976, Y  +375.387, Z    +0.000, E1    +4.229, E3 +60742.466}
SPL {X  -159.990, Y  +379.485, Z    +0.000, E1    +0.028, E3 +60742.511}
SPL {X  -159.990, Y  +381.270, Z    +0.000, E1    -3.383, E3 +60742.528}
SPL {X  -159.990, Y  +386.246, Z    +0.000, E1   -14.704, E3 +60742.686}
SPL {X  -159.990, Y  +394.075, Z    +0.000, E1   -32.836, E3 +60743.246}
SPL {X  -159.990, Y  +405.152, Z    +0.000, E1   -50.697, E3 +60744.671}
SPL {X  -159.990, Y  +423.293, Z    +0.000, E1   -63.280, E3 +60748.672}
SPL {X  -159.990, Y  +493.649, Z    +0.000, E1   -71.671, E3 +60774.376}
SPL {X  -159.990, Y  +662.531, Z    +0.000, E1   -73.010, E3 +60861.199}
SPL {X  -159.805, Y  +684.185, Z    +0.000, E1   -72.979, E3 +60875.483}
SPL {X  -158.295, Y  +699.729, Z    +0.000, E1   -72.830, E3 +60887.153}
SPL {X  -155.857, Y  +712.630, Z    +0.000, E1   -72.572, E3 +60898.082}
SPL {X  -153.206, Y  +722.596, Z    +0.000, E1   -72.287, E3 +60907.263}
SPL {X  -150.445, Y  +730.933, Z    +0.000, E1   -71.979, E3 +60915.474}
SPL {X  -147.389, Y  +738.737, Z    +0.000, E1   -71.634, E3 +60923.546}
SPL {X  -144.044, Y  +746.129, Z    +0.000, E1   -71.236, E3 +60931.541}
SPL {X  -140.684, Y  +752.689, Z    +0.000, E1   -70.820, E3 +60938.916}
SPL {X  -136.099, Y  +760.606, Z    +0.000, E1   -70.253, E3 +60948.071}
SPL {X  -131.456, Y  +767.693, Z    +0.000, E1   -69.587, E3 +60956.583}
SPL {X  -127.440, Y  +773.226, Z    +0.000, E1   -69.006, E3 +60963.267}
SPL {X  -123.127, Y  +778.659, Z    +0.000, E1   -68.349, E3 +60969.809}
SPL {X   -80.879, Y  +814.541, Z    +0.000, E1   -55.704, E3 +61092.713}
ENDSPLINE

SPLINE
SPL {X  -125.518, Y  +775.707, Z    +0.000, E1   -52.189, E3 +61264.190}
SPL {X  -150.797, Y  +729.951, Z    +0.000, E1   -39.777, E3 +61286.925}
SPL {X  -157.402, Y  +705.160, Z    +0.000, E1   -26.108, E3 +61291.877}
SPL {X  -159.480, Y  +689.270, Z    +0.000, E1   -14.023, E3 +61293.443}
SPL {X  -159.986, Y  +677.650, Z    +0.000, E1    -3.291, E3 +61293.937}
SPL {X  -159.990, Y  +674.500, Z    +0.000, E1    +0.000, E3 +61293.968}
SPL {X  -159.990, Y  +672.716, Z    +0.000, E1    +3.405, E3 +61293.984}
SPL {X  -159.990, Y  +668.521, Z    +0.000, E1   +13.007, E3 +61294.103}
SPL {X  -159.990, Y  +662.839, Z    +0.000, E1   +26.519, E3 +61294.445}
SPL {X  -159.990, Y  +653.836, Z    +0.000, E1   +43.967, E3 +61295.376}
SPL {X  -159.990, Y  +641.022, Z    +0.000, E1   +57.726, E3 +61297.685}
SPL {X  -159.990, Y  +617.987, Z    +0.000, E1   +67.134, E3 +61303.580}
SPL {X  -159.990, Y  +532.407, Z    +0.000, E1   +73.084, E3 +61334.487}
SPL {X  -159.990, Y  +390.607, Z    +0.000, E1   +73.632, E3 +61406.023}
SPL {X  -159.886, Y  +371.742, Z    +0.000, E1   +73.650, E3 +61417.810}
SPL {X  -157.928, Y  +351.899, Z    +0.000, E1   +73.451, E3 +61432.243}
ENDSPLINE

SPLINE
SPL {X  -159.990, Y  +380.170, Z    +0.000, E1   +69.785, E3 +61448.384}
ENDSPLINE

SPLINE
SPL {X  -158.227, Y  +353.814, Z    +0.000, E1   +70.663, E3 +61460.277}
SPL {X  -155.560, Y  +340.111, Z    +0.000, E1   +70.976, E3 +61467.299}
SPL {X  -151.918, Y  +327.322, Z    +0.000, E1   +71.266, E3 +61473.643}
SPL {X  -144.697, Y  +309.238, Z    +0.000, E1   +71.848, E3 +61480.592}
SPL {X  -140.298, Y  +300.601, Z    +0.000, E1   +71.461, E3 +61488.880}
SPL {X  -135.903, Y  +293.078, Z    +0.000, E1   +70.930, E3 +61497.417}
SPL {X  -130.487, Y  +284.926, Z    +0.000, E1   +70.202, E3 +61506.977}
SPL {X  -125.807, Y  +278.659, Z    +0.000, E1   +69.508, E3 +61514.433}
SPL {X  -122.967, Y  +275.148, Z    +0.000, E1   +69.053, E3 +61518.602}
SPL {X  -121.236, Y  +273.103, Z    +0.000, E1   +68.779, E3 +61520.988}
SPL {X   -84.117, Y  +241.407, Z    +0.000, E1   +58.224, E3 +61610.693}
ENDSPLINE

SPLINE
SPL {X  -116.986, Y  +268.362, Z    +0.000, E1   +53.233, E3 +61804.609}
SPL {X  -146.319, Y  +312.789, Z    +0.000, E1   +44.152, E3 +61835.075}
SPL {X  -157.053, Y  +346.986, Z    +0.000, E1   +27.437, E3 +61843.106}
SPL {X  -159.518, Y  +365.226, Z    +0.000, E1   +13.562, E3 +61844.972}
SPL {X  -159.976, Y  +375.387, Z    +0.000, E1    +4.229, E3 +61845.407}
SPL {X  -159.990, Y  +379.485, Z    +0.000, E1    +0.028, E3 +61845.452}
SPL {X  -159.990, Y  +381.270, Z    +0.000, E1    -3.383, E3 +61845.469}
SPL {X  -159.990, Y  +386.246, Z    +0.000, E1   -14.704, E3 +61845.627}
SPL {X  -159.990, Y  +394.075, Z    +0.000, E1   -32.836, E3 +61846.188}
SPL {X  -159.990, Y  +405.152, Z    +0.000, E1   -50.697, E3 +61847.612}
SPL {X  -159.990, Y  +423.293, Z    +0.000, E1   -63.280, E3 +61851.613}
SPL {X  -159.990, Y  +493.649, Z    +0.000, E1   -71.671, E3 +61877.317}
SPL {X  -159.990, Y  +662.531, Z    +0.000, E1   -73.010, E3 +61964.140}
SPL {X  -159.805, Y  +684.185, Z    +0.000, E1   -72.979, E3 +61978.424}
SPL {X  -158.295, Y  +699.729, Z    +0.000, E1   -72.830, E3 +61990.095}
SPL {X  -155.857, Y  +712.630, Z    +0.000, E1   -72.572, E3 +62001.024}
SPL {X  -153.206, Y  +722.596, Z    +0.000, E1   -72.287, E3 +62010.204}
SPL {X  -150.445, Y  +730.933, Z    +0.000, E1   -71.979, E3 +62018.415}
SPL {X  -147.389, Y  +738.737, Z    +0.000, E1   -71.634, E3 +62026.487}
SPL {X  -144.044, Y  +746.129, Z    +0.000, E1   -71.236, E3 +62034.482}
SPL {X  -140.684, Y  +752.689, Z    +0.000, E1   -70.820, E3 +62041.857}
SPL {X  -136.099, Y  +760.606, Z    +0.000, E1   -70.253, E3 +62051.013}
SPL {X  -131.456, Y  +767.693, Z    +0.000, E1   -69.587, E3 +62059.524}
SPL {X  -127.440, Y  +773.226, Z    +0.000, E1   -69.006, E3 +62066.208}
SPL {X  -123.127, Y  +778.659, Z    +0.000, E1   -68.349, E3 +62072.750}
SPL {X   -80.879, Y  +814.541, Z    +0.000, E1   -55.704, E3 +62195.654}
ENDSPLINE

SPLINE
SPL {X  -125.518, Y  +775.707, Z    +0.000, E1   -52.189, E3 +62367.132}
SPL {X  -150.797, Y  +729.951, Z    +0.000, E1   -39.777, E3 +62389.866}
SPL {X  -158.456, Y  +698.602, Z    +0.000, E1   -21.523, E3 +62395.569}
SPL {X  -159.738, Y  +685.469, Z    +0.000, E1   -10.595, E3 +62396.623}
SPL {X  -159.986, Y  +677.650, Z    +0.000, E1    -3.291, E3 +62396.878}
SPL {X  -159.990, Y  +674.500, Z    +0.000, E1    +0.000, E3 +62396.909}
SPL {X  -159.990, Y  +672.716, Z    +0.000, E1    +3.405, E3 +62396.925}
SPL {X  -159.990, Y  +668.521, Z    +0.000, E1   +13.007, E3 +62397.044}
SPL {X  -159.990, Y  +662.839, Z    +0.000, E1   +26.519, E3 +62397.387}
SPL {X  -159.990, Y  +653.836, Z    +0.000, E1   +43.967, E3 +62398.317}
SPL {X  -159.990, Y  +641.022, Z    +0.000, E1   +57.726, E3 +62400.626}
SPL {X  -159.990, Y  +617.987, Z    +0.000, E1   +67.134, E3 +62406.521}
SPL {X  -159.990, Y  +532.407, Z    +0.000, E1   +73.084, E3 +62437.428}
SPL {X  -159.990, Y  +382.957, Z    +0.000, E1   +73.647, E3 +62513.688}
SPL {X  -159.615, Y  +366.548, Z    +0.000, E1   +73.602, E3 +62524.330}
SPL {X  -157.928, Y  +351.899, Z    +0.000, E1   +73.451, E3 +62535.184}
ENDSPLINE

SPLINE
SPL {X  -159.990, Y  +380.170, Z    +0.000, E1   +69.785, E3 +62551.325}
ENDSPLINE

SPLINE
SPL {X  -158.227, Y  +353.814, Z    +0.000, E1   +70.663, E3 +62563.218}
SPL {X  -154.257, Y  +335.055, Z    +0.000, E1   +71.089, E3 +62572.846}
SPL {X  -148.153, Y  +317.104, Z    +0.000, E1   +71.658, E3 +62579.992}
SPL {X  -143.479, Y  +306.716, Z    +0.000, E1   +71.847, E3 +62585.065}
SPL {X  -140.298, Y  +300.601, Z    +0.000, E1   +71.461, E3 +62591.821}
SPL {X  -137.001, Y  +294.872, Z    +0.000, E1   +71.048, E3 +62598.329}
SPL {X  -133.301, Y  +289.026, Z    +0.000, E1   +70.567, E3 +62605.116}
SPL {X  -128.648, Y  +282.387, Z    +0.000, E1   +69.939, E3 +62612.931}
SPL {X  -125.063, Y  +277.720, Z    +0.000, E1   +69.378, E3 +62618.507}
SPL {X  -122.086, Y  +274.099, Z    +0.000, E1   +68.932, E3 +62622.752}
SPL {X   -84.117, Y  +241.407, Z    +0.000, E1   +58.224, E3 +62713.635}
ENDSPLINE

SPLINE
SPL {X  -106.708, Y  +258.294, Z    +0.000, E1   +53.789, E3 +62892.422}
SPL {X  -137.973, Y  +296.505, Z    +0.000, E1   +48.844, E3 +62931.202}
SPL {X  -154.359, Y  +335.426, Z    +0.000, E1   +34.338, E3 +62944.098}
SPL {X  -159.279, Y  +362.429, Z    +0.000, E1   +16.013, E3 +62947.698}
SPL {X  -159.976, Y  +375.387, Z    +0.000, E1    +4.229, E3 +62948.348}
SPL {X  -159.990, Y  +379.485, Z    +0.000, E1    +0.028, E3 +62948.394}
SPL {X  -159.990, Y  +381.270, Z    +0.000, E1    -3.383, E3 +62948.411}
SPL {X  -159.990, Y  +384.811, Z    +0.000, E1   -11.531, E3 +62948.501}
SPL {X  -159.990, Y  +390.180, Z    +0.000, E1   -24.142, E3 +62948.804}
SPL {X  -159.990, Y  +397.074, Z    +0.000, E1   -39.012, E3 +62949.414}
SPL {X  -159.990, Y  +405.152, Z    +0.000, E1   -50.697, E3 +62950.553}
SPL {X  -159.990, Y  +423.293, Z    +0.000, E1   -63.280, E3 +62954.554}
SPL {X  -159.990, Y  +493.649, Z    +0.000, E1   -71.671, E3 +62980.258}
SPL {X  -159.990, Y  +662.531, Z    +0.000, E1   -73.010, E3 +63067.081}
SPL {X  -159.805, Y  +684.185, Z    +0.000, E1   -72.979, E3 +63081.365}
SPL {X  -158.739, Y  +696.464, Z    +0.000, E1   -72.862, E3 +63090.484}
SPL {X  -156.417, Y  +710.124, Z    +0.000, E1   -72.650, E3 +63101.707}
SPL {X  -153.206, Y  +722.596, Z    +0.000, E1   -72.287, E3 +63113.146}
SPL {X  -150.445, Y  +730.933, Z    +0.000, E1   -71.979, E3 +63121.356}
SPL {X  -147.389, Y  +738.737, Z    +0.000, E1   -71.634, E3 +63129.429}
SPL {X  -144.044, Y  +746.129, Z    +0.000, E1   -71.236, E3 +63137.423}
SPL {X  -140.684, Y  +752.689, Z    +0.000, E1   -70.820, E3 +63144.798}
SPL {X  -137.335, Y  +758.572, Z    +0.000, E1   -70.388, E3 +63151.606}
SPL {X  -134.566, Y  +763.037, Z    +0.000, E1   -70.007, E3 +63156.902}
SPL {X  -131.456, Y  +767.693, Z    +0.000, E1   -69.587, E3 +63162.465}
SPL {X  -127.440, Y  +773.226, Z    +0.000, E1   -69.006, E3 +63169.149}
SPL {X  -123.127, Y  +778.659, Z    +0.000, E1   -68.349, E3 +63175.691}
SPL {X   -80.879, Y  +814.541, Z    +0.000, E1   -55.704, E3 +63298.595}
ENDSPLINE

SPLINE
SPL {X  -125.518, Y  +775.707, Z    +0.000, E1   -52.189, E3 +63470.073}
SPL {X  -144.748, Y  +744.653, Z    +0.000, E1   -45.208, E3 +63488.269}
SPL {X  -153.147, Y  +722.791, Z    +0.000, E1   -36.417, E3 +63494.664}
SPL {X  -157.402, Y  +705.160, Z    +0.000, E1   -26.108, E3 +63497.759}
SPL {X  -159.480, Y  +689.270, Z    +0.000, E1   -14.023, E3 +63499.325}
SPL {X  -159.986, Y  +677.650, Z    +0.000, E1    -3.291, E3 +63499.819}
SPL {X  -159.990, Y  +674.500, Z    +0.000, E1    +0.000, E3 +63499.850}
SPL {X  -159.990, Y  +672.716, Z    +0.000, E1    +3.405, E3 +63499.866}
SPL {X  -159.990, Y  +668.521, Z    +0.000, E1   +13.007, E3 +63499.985}
SPL {X  -159.990, Y  +662.839, Z    +0.000, E1   +26.519, E3 +63500.328}
SPL {X  -159.990, Y  +653.836, Z    +0.000, E1   +43.967, E3 +63501.258}
SPL {X  -159.990, Y  +641.022, Z    +0.000, E1   +57.726, E3 +63503.567}
SPL {X  -159.990, Y  +617.987, Z    +0.000, E1   +67.134, E3 +63509.463}
SPL {X  -159.990, Y  +532.407, Z    +0.000, E1   +73.084, E3 +63540.369}
SPL {X  -159.990, Y  +382.957, Z    +0.000, E1   +73.647, E3 +63616.629}
SPL {X  -159.615, Y  +366.548, Z    +0.000, E1   +73.602, E3 +63627.271}
SPL {X  -157.928, Y  +351.899, Z    +0.000, E1   +73.451, E3 +63638.126}
ENDSPLINE

SPLINE
SPL {X  -159.990, Y  +380.170, Z    +0.000, E1   +69.785, E3 +63654.266}
ENDSPLINE

SPLINE
SPL {X  -158.227, Y  +353.814, Z    +0.000, E1   +70.663, E3 +63666.159}
SPL {X  -155.560, Y  +340.111, Z    +0.000, E1   +70.976, E3 +63673.181}
SPL {X  -151.918, Y  +327.322, Z    +0.000, E1   +71.266, E3 +63679.525}
SPL {X  -144.697, Y  +309.238, Z    +0.000, E1   +71.848, E3 +63686.475}
SPL {X  -140.298, Y  +300.601, Z    +0.000, E1   +71.461, E3 +63694.762}
SPL {X  -135.903, Y  +293.078, Z    +0.000, E1   +70.930, E3 +63703.300}
SPL {X  -130.487, Y  +284.926, Z    +0.000, E1   +70.202, E3 +63712.859}
SPL {X  -125.807, Y  +278.659, Z    +0.000, E1   +69.508, E3 +63720.316}
SPL {X  -122.967, Y  +275.148, Z    +0.000, E1   +69.053, E3 +63724.484}
SPL {X  -121.236, Y  +273.103, Z    +0.000, E1   +68.779, E3 +63726.870}
SPL {X   -84.117, Y  +241.407, Z    +0.000, E1   +58.224, E3 +63816.576}
ENDSPLINE

SPLINE
SPL {X  -106.708, Y  +258.294, Z    +0.000, E1   +53.789, E3 +63995.363}
SPL {X  -137.973, Y  +296.505, Z    +0.000, E1   +48.844, E3 +64034.143}
SPL {X  -150.692, Y  +323.752, Z    +0.000, E1   +39.895, E3 +64044.509}
SPL {X  -157.053, Y  +346.986, Z    +0.000, E1   +27.437, E3 +64048.989}
SPL {X  -159.518, Y  +365.226, Z    +0.000, E1   +13.562, E3 +64050.854}
SPL {X  -159.976, Y  +375.387, Z    +0.000, E1    +4.229, E3 +64051.290}
SPL {X  -159.990, Y  +379.485, Z    +0.000, E1    +0.028, E3 +64051.335}
SPL {X  -159.990, Y  +381.270, Z    +0.000, E1    -3.383, E3 +64051.352}
SPL {X  -159.990, Y  +384.811, Z    +0.000, E1   -11.531, E3 +64051.442}
SPL {X  -159.990, Y  +390.180, Z    +0.000, E1   -24.142, E3 +64051.745}
SPL {X  -159.990, Y  +397.074, Z    +0.000, E1   -39.012, E3 +64052.355}
SPL {X  -159.990, Y  +405.152, Z    +0.000, E1   -50.697, E3 +64053.494}
SPL {X  -159.990, Y  +423.293, Z    +0.000, E1   -63.280, E3 +64057.496}
SPL {X  -159.990, Y  +493.649, Z    +0.000, E1   -71.671, E3 +64083.199}
SPL {X  -159.990, Y  +662.531, Z    +0.000, E1   -73.010, E3 +64170.023}
SPL {X  -159.805, Y  +684.185, Z    +0.000, E1   -72.979, E3 +64184.307}
SPL {X  -158.739, Y  +696.464, Z    +0.000, E1   -72.862, E3 +64193.425}
SPL {X  -156.417, Y  +710.124, Z    +0.000, E1   -72.650, E3 +64204.649}
SPL {X  -153.206, Y  +722.596, Z    +0.000, E1   -72.287, E3 +64216.087}
SPL {X  -150.445, Y  +730.933, Z    +0.000, E1   -71.979, E3 +64224.297}
SPL {X  -147.389, Y  +738.737, Z    +0.000, E1   -71.634, E3 +64232.370}
SPL {X  -144.044, Y  +746.129, Z    +0.000, E1   -71.236, E3 +64240.364}
SPL {X  -140.684, Y  +752.689, Z    +0.000, E1   -70.820, E3 +64247.740}
SPL {X  -137.335, Y  +758.572, Z    +0.000, E1   -70.388, E3 +64254.547}
SPL {X  -133.651, Y  +764.444, Z    +0.000, E1   -69.897, E3 +64261.499}
SPL {X  -129.492, Y  +770.461, Z    +0.000, E1   -69.311, E3 +64268.739}
SPL {X  -125.168, Y  +776.148, Z    +0.000, E1   -68.666, E3 +64275.615}
SPL {X  -122.036, Y  +779.960, Z    +0.000, E1   -68.144, E3 +64280.219}
SPL {X   -80.879, Y  +814.541, Z    +0.000, E1   -55.704, E3 +64401.536}
ENDSPLINE

SPLINE
SPL {X  -125.518, Y  +775.707, Z    +0.000, E1   -52.189, E3 +64573.014}
SPL {X  -144.748, Y  +744.653, Z    +0.000, E1   -45.208, E3 +64591.210}
SPL {X  -153.147, Y  +722.791, Z    +0.000, E1   -36.417, E3 +64597.605}
SPL {X  -158.456, Y  +698.602, Z    +0.000, E1   -21.523, E3 +64601.451}
SPL {X  -159.738, Y  +685.469, Z    +0.000, E1   -10.595, E3 +64602.506}
SPL {X  -159.986, Y  +677.650, Z    +0.000, E1    -3.291, E3 +64602.761}
SPL {X  -159.990, Y  +674.500, Z    +0.000, E1    +0.000, E3 +64602.791}
SPL {X  -159.990, Y  +672.716, Z    +0.000, E1    +3.405, E3 +64602.808}
SPL {X  -159.990, Y  +668.521, Z    +0.000, E1   +13.007, E3 +64602.927}
SPL {X  -159.990, Y  +662.839, Z    +0.000, E1   +26.519, E3 +64603.269}
SPL {X  -159.990, Y  +653.836, Z    +0.000, E1   +43.967, E3 +64604.199}
SPL {X  -159.990, Y  +641.022, Z    +0.000, E1   +57.726, E3 +64606.508}
SPL {X  -159.990, Y  +617.987, Z    +0.000, E1   +67.134, E3 +64612.404}
SPL {X  -159.990, Y  +532.407, Z    +0.000, E1   +73.084, E3 +64643.310}
SPL {X  -159.990, Y  +382.957, Z    +0.000, E1   +73.647, E3 +64719.570}
SPL {X  -159.615, Y  +366.548, Z    +0.000, E1   +73.602, E3 +64730.212}
SPL {X  -157.928, Y  +351.899, Z    +0.000, E1   +73.451, E3 +64741.067}
ENDSPLINE

SPLINE
SPL {X  -159.990, Y  +380.170, Z    +0.000, E1   +69.785, E3 +64757.207}
ENDSPLINE

SPLINE
SPL {X  -158.227, Y  +353.814, Z    +0.000, E1   +70.663, E3 +64769.101}
SPL {X  -155.560, Y  +340.111, Z    +0.000, E1   +70.976, E3 +64776.123}
SPL {X  -151.918, Y  +327.322, Z    +0.000, E1   +71.266, E3 +64782.466}
SPL {X  -144.697, Y  +309.238, Z    +0.000, E1   +71.848, E3 +64789.416}
SPL {X  -140.298, Y  +300.601, Z    +0.000, E1   +71.461, E3 +64797.703}
SPL {X  -135.903, Y  +293.078, Z    +0.000, E1   +70.930, E3 +64806.241}
SPL {X  -132.382, Y  +287.656, Z    +0.000, E1   +70.425, E3 +64812.633}
SPL {X  -128.648, Y  +282.387, Z    +0.000, E1   +69.939, E3 +64818.813}
SPL {X  -125.063, Y  +277.720, Z    +0.000, E1   +69.378, E3 +64824.389}
SPL {X  -122.086, Y  +274.099, Z    +0.000, E1   +68.932, E3 +64828.634}
SPL {X   -84.117, Y  +241.407, Z    +0.000, E1   +58.224, E3 +64919.517}
ENDSPLINE

SPLINE
SPL {X  -116.986, Y  +268.362, Z    +0.000, E1   +53.233, E3 +65113.432}
SPL {X  -146.319, Y  +312.789, Z    +0.000, E1   +44.152, E3 +65143.899}
SPL {X  -155.980, Y  +341.904, Z    +0.000, E1   +30.583, E3 +65151.194}
SPL {X  -159.279, Y  +362.429, Z    +0.000, E1   +16.013, E3 +65153.580}
SPL {X  -159.976, Y  +375.387, Z    +0.000, E1    +4.229, E3 +65154.231}
SPL {X  -159.990, Y  +379.485, Z    +0.000, E1    +0.028, E3 +65154.276}
SPL {X  -159.990, Y  +381.270, Z    +0.000, E1    -3.383, E3 +65154.293}
SPL {X  -159.990, Y  +386.246, Z    +0.000, E1   -14.704, E3 +65154.450}
SPL {X  -159.990, Y  +394.075, Z    +0.000, E1   -32.836, E3 +65155.011}
SPL {X  -159.990, Y  +405.152, Z    +0.000, E1   -50.697, E3 +65156.435}
SPL {X  -159.990, Y  +423.293, Z    +0.000, E1   -63.280, E3 +65160.437}
SPL {X  -159.990, Y  +493.649, Z    +0.000, E1   -71.671, E3 +65186.141}
SPL {X  -159.990, Y  +662.531, Z    +0.000, E1   -73.010, E3 +65272.964}
SPL {X  -159.805, Y  +684.185, Z    +0.000, E1   -72.979, E3 +65287.248}
SPL {X  -158.295, Y  +699.729, Z    +0.000, E1   -72.830, E3 +65298.918}
SPL {X  -155.857, Y  +712.630, Z    +0.000, E1   -72.572, E3 +65309.847}
SPL {X  -153.206, Y  +722.596, Z    +0.000, E1   -72.287, E3 +65319.028}
SPL {X  -150.445, Y  +730.933, Z    +0.000, E1   -71.979, E3 +65327.238}
SPL {X  -147.389, Y  +738.737, Z    +0.000, E1   -71.634, E3 +65335.311}
SPL {X  -144.044, Y  +746.129, Z    +0.000, E1   -71.236, E3 +65343.305}
SPL {X  -140.684, Y  +752.689, Z    +0.000, E1   -70.820, E3 +65350.681}
SPL {X  -137.335, Y  +758.572, Z    +0.000, E1   -70.388, E3 +65357.488}
SPL {X  -133.651, Y  +764.444, Z    +0.000, E1   -69.897, E3 +65364.440}
SPL {X  -129.492, Y  +770.461, Z    +0.000, E1   -69.311, E3 +65371.680}
SPL {X  -125.168, Y  +776.148, Z    +0.000, E1   -68.666, E3 +65378.557}
SPL {X  -122.036, Y  +779.960, Z    +0.000, E1   -68.144, E3 +65383.160}
SPL {X   -80.879, Y  +814.541, Z    +0.000, E1   -55.704, E3 +65504.478}
ENDSPLINE

SPLINE
SPL {X  -125.518, Y  +775.707, Z    +0.000, E1   -52.189, E3 +65675.955}
SPL {X  -144.748, Y  +744.653, Z    +0.000, E1   -45.208, E3 +65694.151}
SPL {X  -153.147, Y  +722.791, Z    +0.000, E1   -36.417, E3 +65700.547}
SPL {X  -157.402, Y  +705.160, Z    +0.000, E1   -26.108, E3 +65703.642}
SPL {X  -159.480, Y  +689.270, Z    +0.000, E1   -14.023, E3 +65705.208}
SPL {X  -159.986, Y  +677.650, Z    +0.000, E1    -3.291, E3 +65705.702}
SPL {X  -159.990, Y  +674.500, Z    +0.000, E1    +0.000, E3 +65705.732}
SPL {X  -159.990, Y  +672.716, Z    +0.000, E1    +3.405, E3 +65705.749}
SPL {X  -159.990, Y  +668.521, Z    +0.000, E1   +13.007, E3 +65705.868}
SPL {X  -159.990, Y  +664.286, Z    +0.000, E1   +23.338, E3 +65706.099}
SPL {X  -159.990, Y  +658.431, Z    +0.000, E1   +35.998, E3 +65706.594}
SPL {X  -159.990, Y  +650.524, Z    +0.000, E1   +48.779, E3 +65707.582}
SPL {X  -159.990, Y  +641.022, Z    +0.000, E1   +57.726, E3 +65709.449}
SPL {X  -159.990, Y  +617.987, Z    +0.000, E1   +67.134, E3 +65715.345}
SPL {X  -159.990, Y  +532.407, Z    +0.000, E1   +73.084, E3 +65746.252}
SPL {X  -159.990, Y  +382.957, Z    +0.000, E1   +73.647, E3 +65822.511}
SPL {X  -159.615, Y  +366.548, Z    +0.000, E1   +73.602, E3 +65833.154}
SPL {X  -157.928, Y  +351.899, Z    +0.000, E1   +73.451, E3 +65844.008}
ENDSPLINE

SPLINE
SPL {X  -159.990, Y  +387.996, Z    +0.000, E1   +69.509, E3 +65856.438}
ENDSPLINE

SPLINE
SPL {X  -159.889, Y  +371.819, Z    +0.000, E1   +70.046, E3 +65864.165}
SPL {X  -158.227, Y  +353.814, Z    +0.000, E1   +70.663, E3 +65872.042}
SPL {X  -154.257, Y  +335.055, Z    +0.000, E1   +71.089, E3 +65881.670}
SPL {X  -148.153, Y  +317.104, Z    +0.000, E1   +71.658, E3 +65888.815}
SPL {X  -143.479, Y  +306.716, Z    +0.000, E1   +71.847, E3 +65893.889}
SPL {X  -140.298, Y  +300.601, Z    +0.000, E1   +71.461, E3 +65900.644}
SPL {X  -135.903, Y  +293.078, Z    +0.000, E1   +70.930, E3 +65909.182}
SPL {X  -130.487, Y  +284.926, Z    +0.000, E1   +70.202, E3 +65918.741}
SPL {X  -125.807, Y  +278.659, Z    +0.000, E1   +69.508, E3 +65926.198}
SPL {X  -122.967, Y  +275.148, Z    +0.000, E1   +69.053, E3 +65930.367}
SPL {X  -121.236, Y  +273.103, Z    +0.000, E1   +68.779, E3 +65932.752}
SPL {X   -84.117, Y  +241.407, Z    +0.000, E1   +58.224, E3 +66022.458}
ENDSPLINE

SPLINE
SPL {X  -116.986, Y  +268.362, Z    +0.000, E1   +53.233, E3 +66216.374}
SPL {X  -146.319, Y  +312.789, Z    +0.000, E1   +44.152, E3 +66246.840}
SPL {X  -157.053, Y  +346.986, Z    +0.000, E1   +27.437, E3 +66254.871}
SPL {X  -159.518, Y  +365.226, Z    +0.000, E1   +13.562, E3 +66256.736}
SPL {X  -159.976, Y  +375.387, Z    +0.000, E1    +4.229, E3 +66257.172}
SPL {X  -159.990, Y  +379.485, Z    +0.000, E1    +0.028, E3 +66257.217}
SPL {X  -159.990, Y  +381.270, Z    +0.000, E1    -3.383, E3 +66257.234}
SPL {X  -159.990, Y  +386.246, Z    +0.000, E1   -14.704, E3 +66257.392}
SPL {X  -159.990, Y  +394.075, Z    +0.000, E1   -32.836, E3 +66257.952}
SPL {X  -159.990, Y  +405.152, Z    +0.000, E1   -50.697, E3 +66259.377}
SPL {X  -159.990, Y  +423.293, Z    +0.000, E1   -63.280, E3 +66263.378}
SPL {X  -159.990, Y  +493.649, Z    +0.000, E1   -71.671, E3 +66289.082}
SPL {X  -159.990, Y  +662.531, Z    +0.000, E1   -73.010, E3 +66375.905}
SPL {X  -159.805, Y  +684.185, Z    +0.000, E1   -72.979, E3 +66390.189}
SPL {X  -158.295, Y  +699.729, Z    +0.000, E1   -72.830, E3 +66401.859}
SPL {X  -155.857, Y  +712.630, Z    +0.000, E1   -72.572, E3 +66412.788}
SPL {X  -153.206, Y  +722.596, Z    +0.000, E1   -72.287, E3 +66421.969}
SPL {X  -150.445, Y  +730.933, Z    +0.000, E1   -71.979, E3 +66430.179}
SPL {X  -147.389, Y  +738.737, Z    +0.000, E1   -71.634, E3 +66438.252}
SPL {X  -144.044, Y  +746.129, Z    +0.000, E1   -71.236, E3 +66446.247}
SPL {X  -140.684, Y  +752.689, Z    +0.000, E1   -70.820, E3 +66453.622}
SPL {X  -136.099, Y  +760.606, Z    +0.000, E1   -70.253, E3 +66462.777}
SPL {X  -131.456, Y  +767.693, Z    +0.000, E1   -69.587, E3 +66471.289}
SPL {X  -127.440, Y  +773.226, Z    +0.000, E1   -69.006, E3 +66477.973}
SPL {X  -123.127, Y  +778.659, Z    +0.000, E1   -68.349, E3 +66484.515}
SPL {X   -80.879, Y  +814.541, Z    +0.000, E1   -55.704, E3 +66607.419}
ENDSPLINE

SPLINE
SPL {X  -125.518, Y  +775.707, Z    +0.000, E1   -52.189, E3 +66778.896}
SPL {X  -150.797, Y  +729.951, Z    +0.000, E1   -39.777, E3 +66801.631}
SPL {X  -158.456, Y  +698.602, Z    +0.000, E1   -21.523, E3 +66807.334}
SPL {X  -159.738, Y  +685.469, Z    +0.000, E1   -10.595, E3 +66808.388}
SPL {X  -159.986, Y  +677.650, Z    +0.000, E1    -3.291, E3 +66808.643}
SPL {X  -159.990, Y  +674.500, Z    +0.000, E1    +0.000, E3 +66808.673}
SPL {X  -159.990, Y  +672.716, Z    +0.000, E1    +3.405, E3 +66808.690}
SPL {X  -159.990, Y  +668.521, Z    +0.000, E1   +13.007, E3 +66808.809}
SPL {X  -159.990, Y  +662.839, Z    +0.000, E1   +26.519, E3 +66809.151}
SPL {X  -159.990, Y  +653.836, Z    +0.000, E1   +43.967, E3 +66810.082}
SPL {X  -159.990, Y  +641.022, Z    +0.000, E1   +57.726, E3 +66812.391}
SPL {X  -159.990, Y  +617.987, Z    +0.000, E1   +67.134, E3 +66818.286}
SPL {X  -159.990, Y  +532.407, Z    +0.000, E1   +73.084, E3 +66849.193}
SPL {X  -159.990, Y  +382.957, Z    +0.000, E1   +73.647, E3 +66925.452}
SPL {X  -159.615, Y  +366.548, Z    +0.000, E1   +73.602, E3 +66936.095}
SPL {X  -157.928, Y  +351.899, Z    +0.000, E1   +73.451, E3 +66946.949}
ENDSPLINE

SPLINE
SPL {X  -159.990, Y  +380.170, Z    +0.000, E1   +69.785, E3 +66963.089}
ENDSPLINE

SPLINE
SPL {X  -158.227, Y  +353.814, Z    +0.000, E1   +70.663, E3 +66974.983}
SPL {X  -154.257, Y  +335.055, Z    +0.000, E1   +71.089, E3 +66984.611}
SPL {X  -148.153, Y  +317.104, Z    +0.000, E1   +71.658, E3 +66991.756}
SPL {X  -143.479, Y  +306.716, Z    +0.000, E1   +71.847, E3 +66996.830}
SPL {X  -140.298, Y  +300.601, Z    +0.000, E1   +71.461, E3 +67003.586}
SPL {X  -137.001, Y  +294.872, Z    +0.000, E1   +71.048, E3 +67010.094}
SPL {X  -133.301, Y  +289.026, Z    +0.000, E1   +70.567, E3 +67016.880}
SPL {X  -128.648, Y  +282.387, Z    +0.000, E1   +69.939, E3 +67024.696}
SPL {X  -125.063, Y  +277.720, Z    +0.000, E1   +69.378, E3 +67030.271}
SPL {X  -122.086, Y  +274.099, Z    +0.000, E1   +68.932, E3 +67034.517}
SPL {X   -84.117, Y  +241.407, Z    +0.000, E1   +58.224, E3 +67125.399}
ENDSPLINE

SPLINE
SPL {X  -106.708, Y  +258.294, Z    +0.000, E1   +53.789, E3 +67304.186}
SPL {X  -137.973, Y  +296.505, Z    +0.000, E1   +48.844, E3 +67342.966}
SPL {X  -154.359, Y  +335.426, Z    +0.000, E1   +34.338, E3 +67355.862}
SPL {X  -159.279, Y  +362.429, Z    +0.000, E1   +16.013, E3 +67359.462}
SPL {X  -159.976, Y  +375.387, Z    +0.000, E1    +4.229, E3 +67360.113}
SPL {X  -159.990, Y  +379.485, Z    +0.000, E1    +0.028, E3 +67360.158}
SPL {X  -159.990, Y  +381.270, Z    +0.000, E1    -3.383, E3 +67360.175}
SPL {X  -159.990, Y  +386.246, Z    +0.000, E1   -14.704, E3 +67360.333}
SPL {X  -159.990, Y  +394.075, Z    +0.000, E1   -32.836, E3 +67360.894}
SPL {X  -159.990, Y  +405.152, Z    +0.000, E1   -50.697, E3 +67362.318}
SPL {X  -159.990, Y  +423.293, Z    +0.000, E1   -63.280, E3 +67366.319}
SPL {X  -159.990, Y  +493.649, Z    +0.000, E1   -71.671, E3 +67392.023}
SPL {X  -159.990, Y  +662.531, Z    +0.000, E1   -73.010, E3 +67478.846}
SPL {X  -159.805, Y  +684.185, Z    +0.000, E1   -72.979, E3 +67493.130}
SPL {X  -158.739, Y  +696.464, Z    +0.000, E1   -72.862, E3 +67502.249}
SPL {X  -156.417, Y  +710.124, Z    +0.000, E1   -72.650, E3 +67513.472}
SPL {X  -153.206, Y  +722.596, Z    +0.000, E1   -72.287, E3 +67524.910}
SPL {X  -150.445, Y  +730.933, Z    +0.000, E1   -71.979, E3 +67533.121}
SPL {X  -147.389, Y  +738.737, Z    +0.000, E1   -71.634, E3 +67541.193}
SPL {X  -144.044, Y  +746.129, Z    +0.000, E1   -71.236, E3 +67549.188}
SPL {X  -140.684, Y  +752.689, Z    +0.000, E1   -70.820, E3 +67556.563}
SPL {X  -137.335, Y  +758.572, Z    +0.000, E1   -70.388, E3 +67563.370}
SPL {X  -133.651, Y  +764.444, Z    +0.000, E1   -69.897, E3 +67570.322}
SPL {X  -130.650, Y  +768.844, Z    +0.000, E1   -69.455, E3 +67575.644}
SPL {X  -127.440, Y  +773.226, Z    +0.000, E1   -69.006, E3 +67580.914}
SPL {X  -123.127, Y  +778.659, Z    +0.000, E1   -68.349, E3 +67587.456}
SPL {X   -80.879, Y  +814.541, Z    +0.000, E1   -55.704, E3 +67710.360}
ENDSPLINE

SPLINE
SPL {X  -125.518, Y  +775.707, Z    +0.000, E1   -52.189, E3 +67881.837}
SPL {X  -150.797, Y  +729.951, Z    +0.000, E1   -39.777, E3 +67904.572}
SPL {X  -158.456, Y  +698.602, Z    +0.000, E1   -21.523, E3 +67910.275}
SPL {X  -159.738, Y  +685.469, Z    +0.000, E1   -10.595, E3 +67911.329}
SPL {X  -159.986, Y  +677.650, Z    +0.000, E1    -3.291, E3 +67911.584}
SPL {X  -159.990, Y  +674.500, Z    +0.000, E1    +0.000, E3 +67911.615}
SPL {X  -159.990, Y  +672.716, Z    +0.000, E1    +3.405, E3 +67911.631}
SPL {X  -159.990, Y  +668.521, Z    +0.000, E1   +13.007, E3 +67911.750}
SPL {X  -159.990, Y  +662.839, Z    +0.000, E1   +26.519, E3 +67912.093}
SPL {X  -159.990, Y  +653.836, Z    +0.000, E1   +43.967, E3 +67913.023}
SPL {X  -159.990, Y  +641.022, Z    +0.000, E1   +57.726, E3 +67915.332}
SPL {X  -159.990, Y  +617.987, Z    +0.000, E1   +67.134, E3 +67921.227}
SPL {X  -159.990, Y  +532.407, Z    +0.000, E1   +73.084, E3 +67952.134}
SPL {X  -159.990, Y  +382.957, Z    +0.000, E1   +73.647, E3 +68028.394}
SPL {X  -159.615, Y  +366.548, Z    +0.000, E1   +73.602, E3 +68039.036}
SPL {X  -157.928, Y  +351.899, Z    +0.000, E1   +73.451, E3 +68049.890}
ENDSPLINE

SPLINE
SPL {X  -159.990, Y  +380.170, Z    +0.000, E1   +69.785, E3 +68066.031}
ENDSPLINE

SPLINE
SPL {X  -158.227, Y  +353.814, Z    +0.000, E1   +70.663, E3 +68077.924}
SPL {X  -154.257, Y  +335.055, Z    +0.000, E1   +71.089, E3 +68087.552}
SPL {X  -148.153, Y  +317.104, Z    +0.000, E1   +71.658, E3 +68094.698}
SPL {X  -143.479, Y  +306.716, Z    +0.000, E1   +71.847, E3 +68099.771}
SPL {X  -140.298, Y  +300.601, Z    +0.000, E1   +71.461, E3 +68106.527}
SPL {X  -137.001, Y  +294.872, Z    +0.000, E1   +71.048, E3 +68113.035}
SPL {X  -133.301, Y  +289.026, Z    +0.000, E1   +70.567, E3 +68119.822}
SPL {X  -128.648, Y  +282.387, Z    +0.000, E1   +69.939, E3 +68127.637}
SPL {X  -125.063, Y  +277.720, Z    +0.000, E1   +69.378, E3 +68133.213}
SPL {X  -122.086, Y  +274.099, Z    +0.000, E1   +68.932, E3 +68137.458}
SPL {X   -84.117, Y  +241.407, Z    +0.000, E1   +58.224, E3 +68228.341}
ENDSPLINE

SPLINE
SPL {X  -106.708, Y  +258.294, Z    +0.000, E1   +53.789, E3 +68407.127}
SPL {X  -137.973, Y  +296.505, Z    +0.000, E1   +48.844, E3 +68445.908}
SPL {X  -154.359, Y  +335.426, Z    +0.000, E1   +34.338, E3 +68458.804}
SPL {X  -159.279, Y  +362.429, Z    +0.000, E1   +16.013, E3 +68462.404}
SPL {X  -159.976, Y  +375.387, Z    +0.000, E1    +4.229, E3 +68463.054}
SPL {X  -159.990, Y  +379.485, Z    +0.000, E1    +0.028, E3 +68463.099}
SPL {X  -159.990, Y  +381.270, Z    +0.000, E1    -3.383, E3 +68463.117}
SPL {X  -159.990, Y  +384.811, Z    +0.000, E1   -11.531, E3 +68463.207}
SPL {X  -159.990, Y  +388.002, Z    +0.000, E1   -19.281, E3 +68463.357}
SPL {X  -159.990, Y  +394.075, Z    +0.000, E1   -32.836, E3 +68463.835}
SPL {X  -159.990, Y  +405.152, Z    +0.000, E1   -50.697, E3 +68465.259}
SPL {X  -159.990, Y  +423.293, Z    +0.000, E1   -63.280, E3 +68469.260}
SPL {X  -159.990, Y  +493.649, Z    +0.000, E1   -71.671, E3 +68494.964}
SPL {X  -159.990, Y  +662.531, Z    +0.000, E1   -73.010, E3 +68581.787}
SPL {X  -159.805, Y  +684.185, Z    +0.000, E1   -72.979, E3 +68596.071}
SPL {X  -158.739, Y  +696.464, Z    +0.000, E1   -72.862, E3 +68605.190}
SPL {X  -156.417, Y  +710.124, Z    +0.000, E1   -72.650, E3 +68616.413}
SPL {X  -153.206, Y  +722.596, Z    +0.000, E1   -72.287, E3 +68627.851}
SPL {X  -150.445, Y  +730.933, Z    +0.000, E1   -71.979, E3 +68636.062}
SPL {X  -147.389, Y  +738.737, Z    +0.000, E1   -71.634, E3 +68644.135}
SPL {X  -144.044, Y  +746.129, Z    +0.000, E1   -71.236, E3 +68652.129}
SPL {X  -140.684, Y  +752.689, Z    +0.000, E1   -70.820, E3 +68659.504}
SPL {X  -137.335, Y  +758.572, Z    +0.000, E1   -70.388, E3 +68666.311}
SPL {X  -134.566, Y  +763.037, Z    +0.000, E1   -70.007, E3 +68671.608}
SPL {X  -131.456, Y  +767.693, Z    +0.000, E1   -69.587, E3 +68677.171}
SPL {X  -127.440, Y  +773.226, Z    +0.000, E1   -69.006, E3 +68683.855}
SPL {X  -123.127, Y  +778.659, Z    +0.000, E1   -68.349, E3 +68690.397}
SPL {X   -80.879, Y  +814.541, Z    +0.000, E1   -55.704, E3 +68813.301}
ENDSPLINE

SPLINE
SPL {X  -125.518, Y  +775.707, Z    +0.000, E1   -52.189, E3 +68984.779}
SPL {X  -150.797, Y  +729.951, Z    +0.000, E1   -39.777, E3 +69007.514}
SPL {X  -158.456, Y  +698.602, Z    +0.000, E1   -21.523, E3 +69013.216}
SPL {X  -159.738, Y  +685.469, Z    +0.000, E1   -10.595, E3 +69014.271}
SPL {X  -159.986, Y  +677.650, Z    +0.000, E1    -3.291, E3 +69014.525}
SPL {X  -159.990, Y  +674.500, Z    +0.000, E1    +0.000, E3 +69014.556}
SPL {X  -159.990, Y  +672.716, Z    +0.000, E1    +3.405, E3 +69014.572}
SPL {X  -159.990, Y  +668.521, Z    +0.000, E1   +13.007, E3 +69014.691}
SPL {X  -159.990, Y  +664.286, Z    +0.000, E1   +23.338, E3 +69014.923}
SPL {X  -159.990, Y  +658.431, Z    +0.000, E1   +35.998, E3 +69015.417}
SPL {X  -159.990, Y  +650.524, Z    +0.000, E1   +48.779, E3 +69016.406}
SPL {X  -159.990, Y  +641.022, Z    +0.000, E1   +57.726, E3 +69018.273}
SPL {X  -159.990, Y  +617.987, Z    +0.000, E1   +67.134, E3 +69024.168}
SPL {X  -159.990, Y  +532.407, Z    +0.000, E1   +73.084, E3 +69055.075}
SPL {X  -159.990, Y  +390.607, Z    +0.000, E1   +73.632, E3 +69126.611}
SPL {X  -159.886, Y  +371.742, Z    +0.000, E1   +73.650, E3 +69138.398}
SPL {X  -157.928, Y  +351.899, Z    +0.000, E1   +73.451, E3 +69152.832}
ENDSPLINE

SPLINE
SPL {X  -159.990, Y  +380.170, Z    +0.000, E1   +69.785, E3 +69168.972}
ENDSPLINE

SPLINE
SPL {X  -158.227, Y  +353.814, Z    +0.000, E1   +70.663, E3 +69180.865}
SPL {X  -154.257, Y  +335.055, Z    +0.000, E1   +71.089, E3 +69190.493}
SPL {X  -148.153, Y  +317.104, Z    +0.000, E1   +71.658, E3 +69197.639}
SPL {X  -143.479, Y  +306.716, Z    +0.000, E1   +71.847, E3 +69202.712}
SPL {X  -140.298, Y  +300.601, Z    +0.000, E1   +71.461, E3 +69209.468}
SPL {X  -137.001, Y  +294.872, Z    +0.000, E1   +71.048, E3 +69215.976}
SPL {X  -133.301, Y  +289.026, Z    +0.000, E1   +70.567, E3 +69222.763}
SPL {X  -129.603, Y  +283.692, Z    +0.000, E1   +70.051, E3 +69229.063}
SPL {X  -125.807, Y  +278.659, Z    +0.000, E1   +69.508, E3 +69235.022}
SPL {X  -122.086, Y  +274.099, Z    +0.000, E1   +68.932, E3 +69240.399}
SPL {X   -84.117, Y  +241.407, Z    +0.000, E1   +58.224, E3 +69331.282}
ENDSPLINE

SPLINE
SPL {X  -106.708, Y  +258.294, Z    +0.000, E1   +53.789, E3 +69510.069}
SPL {X  -137.973, Y  +296.505, Z    +0.000, E1   +48.844, E3 +69548.849}
SPL {X  -154.359, Y  +335.426, Z    +0.000, E1   +34.338, E3 +69561.745}
SPL {X  -159.279, Y  +362.429, Z    +0.000, E1   +16.013, E3 +69565.345}
SPL {X  -159.976, Y  +375.387, Z    +0.000, E1    +4.229, E3 +69565.996}
SPL {X  -159.990, Y  +379.485, Z    +0.000, E1    +0.028, E3 +69566.041}
SPL {X  -159.990, Y  +381.270, Z    +0.000, E1    -3.383, E3 +69566.058}
SPL {X  -159.990, Y  +386.246, Z    +0.000, E1   -14.704, E3 +69566.215}
SPL {X  -159.990, Y  +394.075, Z    +0.000, E1   -32.836, E3 +69566.776}
SPL {X  -159.990, Y  +405.152, Z    +0.000, E1   -50.697, E3 +69568.200}
SPL {X  -159.990, Y  +423.293, Z    +0.000, E1   -63.280, E3 +69572.201}
SPL {X  -159.990, Y  +493.649, Z    +0.000, E1   -71.671, E3 +69597.905}
SPL {X  -159.990, Y  +662.531, Z    +0.000, E1   -73.010, E3 +69684.728}
SPL {X  -159.805, Y  +684.185, Z    +0.000, E1   -72.979, E3 +69699.012}
SPL {X  -158.295, Y  +699.729, Z    +0.000, E1   -72.830, E3 +69710.683}
SPL {X  -155.857, Y  +712.630, Z    +0.000, E1   -72.572, E3 +69721.612}
SPL {X  -153.206, Y  +722.596, Z    +0.000, E1   -72.287, E3 +69730.793}
SPL {X  -150.445, Y  +730.933, Z    +0.000, E1   -71.979, E3 +69739.003}
SPL {X  -147.389, Y  +738.737, Z    +0.000, E1   -71.634, E3 +69747.076}
SPL {X  -144.044, Y  +746.129, Z    +0.000, E1   -71.236, E3 +69755.070}
SPL {X  -140.684, Y  +752.689, Z    +0.000, E1   -70.820, E3 +69762.445}
SPL {X  -137.335, Y  +758.572, Z    +0.000, E1   -70.388, E3 +69769.253}
SPL {X  -134.566, Y  +763.037, Z    +0.000, E1   -70.007, E3 +69774.549}
SPL {X  -131.456, Y  +767.693, Z    +0.000, E1   -69.587, E3 +69780.113}
SPL {X  -127.440, Y  +773.226, Z    +0.000, E1   -69.006, E3 +69786.796}
SPL {X  -123.127, Y  +778.659, Z    +0.000, E1   -68.349, E3 +69793.338}
SPL {X   -80.879, Y  +814.541, Z    +0.000, E1   -55.704, E3 +69916.242}
ENDSPLINE

SPLINE
SPL {X  -125.518, Y  +775.707, Z    +0.000, E1   -52.189, E3 +70087.720}
SPL {X  -144.748, Y  +744.653, Z    +0.000, E1   -45.208, E3 +70105.916}
SPL {X  -153.147, Y  +722.791, Z    +0.000, E1   -36.417, E3 +70112.311}
SPL {X  -157.402, Y  +705.160, Z    +0.000, E1   -26.108, E3 +70115.407}
SPL {X  -159.480, Y  +689.270, Z    +0.000, E1   -14.023, E3 +70116.972}
SPL {X  -159.986, Y  +677.650, Z    +0.000, E1    -3.291, E3 +70117.467}
SPL {X  -159.990, Y  +674.500, Z    +0.000, E1    +0.000, E3 +70117.497}
SPL {X  -159.990, Y  +672.716, Z    +0.000, E1    +3.405, E3 +70117.513}
SPL {X  -159.990, Y  +668.521, Z    +0.000, E1   +13.007, E3 +70117.633}
SPL {X  -159.990, Y  +664.286, Z    +0.000, E1   +23.338, E3 +70117.864}
SPL {X  -159.990, Y  +658.431, Z    +0.000, E1   +35.998, E3 +70118.359}
SPL {X  -159.990, Y  +650.524, Z    +0.000, E1   +48.779, E3 +70119.347}
SPL {X  -159.990, Y  +641.022, Z    +0.000, E1   +57.726, E3 +70121.214}
SPL {X  -159.990, Y  +617.987, Z    +0.000, E1   +67.134, E3 +70127.110}
SPL {X  -159.990, Y  +532.407, Z    +0.000, E1   +73.084, E3 +70158.016}
SPL {X  -159.990, Y  +390.607, Z    +0.000, E1   +73.632, E3 +70229.552}
SPL {X  -159.886, Y  +371.742, Z    +0.000, E1   +73.650, E3 +70241.339}
SPL {X  -157.928, Y  +351.899, Z    +0.000, E1   +73.451, E3 +70255.773}
ENDSPLINE

SPLINE
SPL {X  -159.990, Y  +380.170, Z    +0.000, E1   +69.785, E3 +70271.913}
ENDSPLINE

SPLINE
SPL {X  -158.227, Y  +353.814, Z    +0.000, E1   +70.663, E3 +70283.806}
SPL {X  -154.257, Y  +335.055, Z    +0.000, E1   +71.089, E3 +70293.434}
SPL {X  -148.153, Y  +317.104, Z    +0.000, E1   +71.658, E3 +70300.580}
SPL {X  -143.479, Y  +306.716, Z    +0.000, E1   +71.847, E3 +70305.654}
SPL {X  -140.298, Y  +300.601, Z    +0.000, E1   +71.461, E3 +70312.409}
SPL {X  -137.001, Y  +294.872, Z    +0.000, E1   +71.048, E3 +70318.917}
SPL {X  -133.301, Y  +289.026, Z    +0.000, E1   +70.567, E3 +70325.704}
SPL {X  -129.603, Y  +283.692, Z    +0.000, E1   +70.051, E3 +70332.004}
SPL {X  -125.807, Y  +278.659, Z    +0.000, E1   +69.508, E3 +70337.963}
SPL {X  -122.086, Y  +274.099, Z    +0.000, E1   +68.932, E3 +70343.340}
SPL {X   -84.117, Y  +241.407, Z    +0.000, E1   +58.224, E3 +70434.223}
ENDSPLINE

SPLINE
SPL {X  -116.986, Y  +268.362, Z    +0.000, E1   +53.233, E3 +70628.138}
SPL {X  -146.319, Y  +312.789, Z    +0.000, E1   +44.152, E3 +70658.604}
SPL {X  -157.053, Y  +346.986, Z    +0.000, E1   +27.437, E3 +70666.636}
SPL {X  -159.518, Y  +365.226, Z    +0.000, E1   +13.562, E3 +70668.501}
SPL {X  -159.976, Y  +375.387, Z    +0.000, E1    +4.229, E3 +70668.937}
SPL {X  -159.990, Y  +379.485, Z    +0.000, E1    +0.028, E3 +70668.982}
SPL {X  -159.990, Y  +381.270, Z    +0.000, E1    -3.383, E3 +70668.999}
SPL {X  -159.990, Y  +384.811, Z    +0.000, E1   -11.531, E3 +70669.089}
SPL {X  -159.990, Y  +388.002, Z    +0.000, E1   -19.281, E3 +70669.239}
SPL {X  -159.990, Y  +394.075, Z    +0.000, E1   -32.836, E3 +70669.717}
SPL {X  -159.990, Y  +405.152, Z    +0.000, E1   -50.697, E3 +70671.141}
SPL {X  -159.990, Y  +423.293, Z    +0.000, E1   -63.280, E3 +70675.143}
SPL {X  -159.990, Y  +493.649, Z    +0.000, E1   -71.671, E3 +70700.847}
SPL {X  -159.990, Y  +654.929, Z    +0.000, E1   -72.988, E3 +70782.796}
SPL {X  -159.990, Y  +668.018, Z    +0.000, E1   -72.989, E3 +70791.289}
SPL {X  -159.805, Y  +684.185, Z    +0.000, E1   -72.979, E3 +70801.954}
SPL {X  -158.295, Y  +699.729, Z    +0.000, E1   -72.830, E3 +70813.624}
SPL {X  -155.857, Y  +712.630, Z    +0.000, E1   -72.572, E3 +70824.553}
SPL {X  -153.206, Y  +722.596, Z    +0.000, E1   -72.287, E3 +70833.734}
SPL {X  -150.445, Y  +730.933, Z    +0.000, E1   -71.979, E3 +70841.944}
SPL {X  -147.389, Y  +738.737, Z    +0.000, E1   -71.634, E3 +70850.017}
SPL {X  -144.044, Y  +746.129, Z    +0.000, E1   -71.236, E3 +70858.011}
SPL {X  -140.684, Y  +752.689, Z    +0.000, E1   -70.820, E3 +70865.387}
SPL {X  -136.099, Y  +760.606, Z    +0.000, E1   -70.253, E3 +70874.542}
SPL {X  -131.456, Y  +767.693, Z    +0.000, E1   -69.587, E3 +70883.054}
SPL {X  -128.507, Y  +771.803, Z    +0.000, E1   -69.145, E3 +70888.036}
SPL {X  -125.168, Y  +776.148, Z    +0.000, E1   -68.666, E3 +70893.262}
SPL {X  -122.036, Y  +779.960, Z    +0.000, E1   -68.144, E3 +70897.866}
SPL {X   -80.879, Y  +814.541, Z    +0.000, E1   -55.704, E3 +71019.184}
ENDSPLINE

SPLINE
SPL {X  -125.518, Y  +775.707, Z    +0.000, E1   -52.189, E3 +71190.661}
SPL {X  -144.748, Y  +744.653, Z    +0.000, E1   -45.208, E3 +71208.857}
SPL {X  -153.147, Y  +722.791, Z    +0.000, E1   -36.417, E3 +71215.252}
SPL {X  -158.456, Y  +698.602, Z    +0.000, E1   -21.523, E3 +71219.099}
SPL {X  -159.738, Y  +685.469, Z    +0.000, E1   -10.595, E3 +71220.153}
SPL {X  -159.986, Y  +677.650, Z    +0.000, E1    -3.291, E3 +71220.408}
SPL {X  -159.990, Y  +674.500, Z    +0.000, E1    +0.000, E3 +71220.438}
SPL {X  -159.990, Y  +672.716, Z    +0.000, E1    +3.405, E3 +71220.455}
SPL {X  -159.990, Y  +668.521, Z    +0.000, E1   +13.007, E3 +71220.574}
SPL {X  -159.990, Y  +664.286, Z    +0.000, E1   +23.338, E3 +71220.805}
SPL {X  -159.990, Y  +658.431, Z    +0.000, E1   +35.998, E3 +71221.300}
SPL {X  -159.990, Y  +650.524, Z    +0.000, E1   +48.779, E3 +71222.288}
SPL {X  -159.990, Y  +641.022, Z    +0.000, E1   +57.726, E3 +71224.155}
SPL {X  -159.990, Y  +617.987, Z    +0.000, E1   +67.134, E3 +71230.051}
SPL {X  -159.990, Y  +532.407, Z    +0.000, E1   +73.084, E3 +71260.957}
SPL {X  -159.990, Y  +382.957, Z    +0.000, E1   +73.647, E3 +71337.217}
SPL {X  -159.615, Y  +366.548, Z    +0.000, E1   +73.602, E3 +71347.859}
SPL {X  -157.928, Y  +351.899, Z    +0.000, E1   +73.451, E3 +71358.714}
ENDSPLINE

SPLINE
SPL {X  -159.990, Y  +380.170, Z    +0.000, E1   +69.785, E3 +71374.854}
ENDSPLINE

SPLINE
SPL {X  -158.227, Y  +353.814, Z    +0.000, E1   +70.663, E3 +71386.748}
SPL {X  -155.560, Y  +340.111, Z    +0.000, E1   +70.976, E3 +71393.770}
SPL {X  -151.918, Y  +327.322, Z    +0.000, E1   +71.266, E3 +71400.113}
SPL {X  -144.697, Y  +309.238, Z    +0.000, E1   +71.848, E3 +71407.063}
SPL {X  -140.298, Y  +300.601, Z    +0.000, E1   +71.461, E3 +71415.350}
SPL {X  -137.001, Y  +294.872, Z    +0.000, E1   +71.048, E3 +71421.859}
SPL {X  -133.301, Y  +289.026, Z    +0.000, E1   +70.567, E3 +71428.645}
SPL {X  -128.648, Y  +282.387, Z    +0.000, E1   +69.939, E3 +71436.460}
SPL {X  -125.063, Y  +277.720, Z    +0.000, E1   +69.378, E3 +71442.036}
SPL {X  -122.086, Y  +274.099, Z    +0.000, E1   +68.932, E3 +71446.281}
SPL {X   -84.117, Y  +241.407, Z    +0.000, E1   +58.224, E3 +71537.164}
ENDSPLINE

SPLINE
SPL {X  -106.708, Y  +258.294, Z    +0.000, E1   +53.789, E3 +71715.951}
SPL {X  -137.973, Y  +296.505, Z    +0.000, E1   +48.844, E3 +71754.731}
SPL {X  -154.359, Y  +335.426, Z    +0.000, E1   +34.338, E3 +71767.627}
SPL {X  -159.279, Y  +362.429, Z    +0.000, E1   +16.013, E3 +71771.227}
SPL {X  -159.976, Y  +375.387, Z    +0.000, E1    +4.229, E3 +71771.878}
SPL {X  -159.990, Y  +379.485, Z    +0.000, E1    +0.028, E3 +71771.923}
SPL {X  -159.990, Y  +381.270, Z    +0.000, E1    -3.383, E3 +71771.940}
SPL {X  -159.990, Y  +384.811, Z    +0.000, E1   -11.531, E3 +71772.030}
SPL {X  -159.990, Y  +390.180, Z    +0.000, E1   -24.142, E3 +71772.333}
SPL {X  -159.990, Y  +397.074, Z    +0.000, E1   -39.012, E3 +71772.943}
SPL {X  -159.990, Y  +405.152, Z    +0.000, E1   -50.697, E3 +71774.082}
SPL {X  -159.990, Y  +423.293, Z    +0.000, E1   -63.280, E3 +71778.084}
SPL {X  -159.990, Y  +493.649, Z    +0.000, E1   -71.671, E3 +71803.788}
SPL {X  -159.990, Y  +662.531, Z    +0.000, E1   -73.010, E3 +71890.611}
SPL {X  -159.805, Y  +684.185, Z    +0.000, E1   -72.979, E3 +71904.895}
SPL {X  -158.295, Y  +699.729, Z    +0.000, E1   -72.830, E3 +71916.565}
SPL {X  -155.857, Y  +712.630, Z    +0.000, E1   -72.572, E3 +71927.494}
SPL {X  -153.206, Y  +722.596, Z    +0.000, E1   -72.287, E3 +71936.675}
SPL {X  -150.445, Y  +730.933, Z    +0.000, E1   -71.979, E3 +71944.885}
SPL {X  -147.389, Y  +738.737, Z    +0.000, E1   -71.634, E3 +71952.958}
SPL {X  -144.044, Y  +746.129, Z    +0.000, E1   -71.236, E3 +71960.952}
SPL {X  -140.684, Y  +752.689, Z    +0.000, E1   -70.820, E3 +71968.328}
SPL {X  -136.099, Y  +760.606, Z    +0.000, E1   -70.253, E3 +71977.483}
SPL {X  -131.456, Y  +767.693, Z    +0.000, E1   -69.587, E3 +71985.995}
SPL {X  -128.507, Y  +771.803, Z    +0.000, E1   -69.145, E3 +71990.977}
SPL {X  -125.168, Y  +776.148, Z    +0.000, E1   -68.666, E3 +71996.204}
SPL {X  -122.036, Y  +779.960, Z    +0.000, E1   -68.144, E3 +72000.807}
SPL {X   -80.879, Y  +814.541, Z    +0.000, E1   -55.704, E3 +72122.125}
ENDSPLINE

SPLINE
SPL {X  -125.518, Y  +775.707, Z    +0.000, E1   -52.189, E3 +72293.602}
SPL {X  -144.748, Y  +744.653, Z    +0.000, E1   -45.208, E3 +72311.798}
SPL {X  -153.147, Y  +722.791, Z    +0.000, E1   -36.417, E3 +72318.194}
SPL {X  -158.456, Y  +698.602, Z    +0.000, E1   -21.523, E3 +72322.040}
SPL {X  -159.738, Y  +685.469, Z    +0.000, E1   -10.595, E3 +72323.094}
SPL {X  -159.986, Y  +677.650, Z    +0.000, E1    -3.291, E3 +72323.349}
SPL {X  -159.990, Y  +674.500, Z    +0.000, E1    +0.000, E3 +72323.379}
SPL {X  -159.990, Y  +672.716, Z    +0.000, E1    +3.405, E3 +72323.396}
SPL {X  -159.990, Y  +668.521, Z    +0.000, E1   +13.007, E3 +72323.515}
SPL {X  -159.990, Y  +664.286, Z    +0.000, E1   +23.338, E3 +72323.746}
SPL {X  -159.990, Y  +658.431, Z    +0.000, E1   +35.998, E3 +72324.241}
SPL {X  -159.990, Y  +650.524, Z    +0.000, E1   +48.779, E3 +72325.229}
SPL {X  -159.990, Y  +641.022, Z    +0.000, E1   +57.726, E3 +72327.096}
SPL {X  -159.990, Y  +617.987, Z    +0.000, E1   +67.134, E3 +72332.992}
SPL {X  -159.990, Y  +532.407, Z    +0.000, E1   +73.084, E3 +72363.899}
SPL {X  -159.990, Y  +382.957, Z    +0.000, E1   +73.647, E3 +72440.158}
SPL {X  -159.615, Y  +366.548, Z    +0.000, E1   +73.602, E3 +72450.801}
SPL {X  -157.928, Y  +351.899, Z    +0.000, E1   +73.451, E3 +72461.655}
ENDSPLINE

SPLINE
SPL {X  -159.990, Y  +380.170, Z    +0.000, E1   +69.785, E3 +72477.795}
ENDSPLINE

SPLINE
SPL {X  -158.227, Y  +353.814, Z    +0.000, E1   +70.663, E3 +72489.689}
SPL {X  -155.560, Y  +340.111, Z    +0.000, E1   +70.976, E3 +72496.711}
SPL {X  -151.918, Y  +327.322, Z    +0.000, E1   +71.266, E3 +72503.054}
SPL {X  -144.697, Y  +309.238, Z    +0.000, E1   +71.848, E3 +72510.004}
SPL {X  -140.298, Y  +300.601, Z    +0.000, E1   +71.461, E3 +72518.292}
SPL {X  -137.001, Y  +294.872, Z    +0.000, E1   +71.048, E3 +72524.800}
SPL {X  -133.301, Y  +289.026, Z    +0.000, E1   +70.567, E3 +72531.586}
SPL {X  -128.648, Y  +282.387, Z    +0.000, E1   +69.939, E3 +72539.402}
SPL {X  -125.063, Y  +277.720, Z    +0.000, E1   +69.378, E3 +72544.977}
SPL {X  -122.086, Y  +274.099, Z    +0.000, E1   +68.932, E3 +72549.223}
SPL {X   -84.117, Y  +241.407, Z    +0.000, E1   +58.224, E3 +72640.105}
ENDSPLINE

SPLINE
SPL {X  -106.708, Y  +258.294, Z    +0.000, E1   +53.789, E3 +72818.892}
SPL {X  -137.973, Y  +296.505, Z    +0.000, E1   +48.844, E3 +72857.672}
SPL {X  -154.359, Y  +335.426, Z    +0.000, E1   +34.338, E3 +72870.568}
SPL {X  -159.279, Y  +362.429, Z    +0.000, E1   +16.013, E3 +72874.168}
SPL {X  -159.976, Y  +375.387, Z    +0.000, E1    +4.229, E3 +72874.819}
SPL {X  -159.990, Y  +379.485, Z    +0.000, E1    +0.028, E3 +72874.864}
SPL {X  -159.990, Y  +381.270, Z    +0.000, E1    -3.383, E3 +72874.881}
SPL {X  -159.990, Y  +384.811, Z    +0.000, E1   -11.531, E3 +72874.971}
SPL {X  -159.990, Y  +390.180, Z    +0.000, E1   -24.142, E3 +72875.274}
SPL {X  -159.990, Y  +397.074, Z    +0.000, E1   -39.012, E3 +72875.884}
SPL {X  -159.990, Y  +405.152, Z    +0.000, E1   -50.697, E3 +72877.024}
SPL {X  -159.990, Y  +423.293, Z    +0.000, E1   -63.280, E3 +72881.025}
SPL {X  -159.990, Y  +493.649, Z    +0.000, E1   -71.671, E3 +72906.729}
SPL {X  -159.990, Y  +662.531, Z    +0.000, E1   -73.010, E3 +72993.552}
SPL {X  -159.805, Y  +684.185, Z    +0.000, E1   -72.979, E3 +73007.836}
SPL {X  -158.739, Y  +696.464, Z    +0.000, E1   -72.862, E3 +73016.955}
SPL {X  -156.417, Y  +710.124, Z    +0.000, E1   -72.650, E3 +73028.178}
SPL {X  -153.206, Y  +722.596, Z    +0.000, E1   -72.287, E3 +73039.616}
SPL {X  -150.445, Y  +730.933, Z    +0.000, E1   -71.979, E3 +73047.827}
SPL {X  -147.389, Y  +738.737, Z    +0.000, E1   -71.634, E3 +73055.899}
SPL {X  -144.044, Y  +746.129, Z    +0.000, E1   -71.236, E3 +73063.894}
SPL {X  -140.684, Y  +752.689, Z    +0.000, E1   -70.820, E3 +73071.269}
SPL {X  -137.335, Y  +758.572, Z    +0.000, E1   -70.388, E3 +73078.076}
SPL {X  -134.566, Y  +763.037, Z    +0.000, E1   -70.007, E3 +73083.372}
SPL {X  -131.456, Y  +767.693, Z    +0.000, E1   -69.587, E3 +73088.936}
SPL {X  -127.440, Y  +773.226, Z    +0.000, E1   -69.006, E3 +73095.620}
SPL {X  -123.127, Y  +778.659, Z    +0.000, E1   -68.349, E3 +73102.162}
SPL {X   -80.879, Y  +814.541, Z    +0.000, E1   -55.704, E3 +73225.066}
ENDSPLINE

SPLINE
SPL {X  -125.518, Y  +775.707, Z    +0.000, E1   -52.189, E3 +73396.543}
SPL {X  -144.748, Y  +744.653, Z    +0.000, E1   -45.208, E3 +73414.739}
SPL {X  -153.147, Y  +722.791, Z    +0.000, E1   -36.417, E3 +73421.135}
SPL {X  -157.402, Y  +705.160, Z    +0.000, E1   -26.108, E3 +73424.230}
SPL {X  -159.480, Y  +689.270, Z    +0.000, E1   -14.023, E3 +73425.796}
SPL {X  -159.986, Y  +677.650, Z    +0.000, E1    -3.291, E3 +73426.290}
SPL {X  -159.990, Y  +674.500, Z    +0.000, E1    +0.000, E3 +73426.320}
SPL {X  -159.990, Y  +672.716, Z    +0.000, E1    +3.405, E3 +73426.337}
SPL {X  -159.990, Y  +668.521, Z    +0.000, E1   +13.007, E3 +73426.456}
SPL {X  -159.990, Y  +662.839, Z    +0.000, E1   +26.519, E3 +73426.798}
SPL {X  -159.990, Y  +653.836, Z    +0.000, E1   +43.967, E3 +73427.729}
SPL {X  -159.990, Y  +641.022, Z    +0.000, E1   +57.726, E3 +73430.038}
SPL {X  -159.990, Y  +617.987, Z    +0.000, E1   +67.134, E3 +73435.933}
SPL {X  -159.990, Y  +532.407, Z    +0.000, E1   +73.084, E3 +73466.840}
SPL {X  -159.990, Y  +382.957, Z    +0.000, E1   +73.647, E3 +73543.099}
SPL {X  -159.615, Y  +366.548, Z    +0.000, E1   +73.602, E3 +73553.742}
SPL {X  -157.928, Y  +351.899, Z    +0.000, E1   +73.451, E3 +73564.596}
ENDSPLINE

SPLINE
SPL {X  -159.990, Y  +380.170, Z    +0.000, E1   +69.785, E3 +73580.736}
ENDSPLINE

SPLINE
SPL {X  -158.227, Y  +353.814, Z    +0.000, E1   +70.663, E3 +73592.630}
SPL {X  -155.560, Y  +340.111, Z    +0.000, E1   +70.976, E3 +73599.652}
SPL {X  -151.918, Y  +327.322, Z    +0.000, E1   +71.266, E3 +73605.996}
SPL {X  -144.697, Y  +309.238, Z    +0.000, E1   +71.848, E3 +73612.945}
SPL {X  -140.298, Y  +300.601, Z    +0.000, E1   +71.461, E3 +73621.233}
SPL {X  -135.903, Y  +293.078, Z    +0.000, E1   +70.930, E3 +73629.770}
SPL {X  -130.487, Y  +284.926, Z    +0.000, E1   +70.202, E3 +73639.330}
SPL {X  -125.807, Y  +278.659, Z    +0.000, E1   +69.508, E3 +73646.786}
SPL {X  -122.967, Y  +275.148, Z    +0.000, E1   +69.053, E3 +73650.955}
SPL {X  -121.236, Y  +273.103, Z    +0.000, E1   +68.779, E3 +73653.341}
SPL {X   -84.117, Y  +241.407, Z    +0.000, E1   +58.224, E3 +73743.046}
ENDSPLINE

SPLINE
SPL {X  -106.708, Y  +258.294, Z    +0.000, E1   +53.789, E3 +73921.833}
SPL {X  -137.973, Y  +296.505, Z    +0.000, E1   +48.844, E3 +73960.613}
SPL {X  -150.692, Y  +323.752, Z    +0.000, E1   +39.895, E3 +73970.979}
SPL {X  -157.053, Y  +346.986, Z    +0.000, E1   +27.437, E3 +73975.459}
SPL {X  -159.518, Y  +365.226, Z    +0.000, E1   +13.562, E3 +73977.325}
SPL {X  -159.976, Y  +375.387, Z    +0.000, E1    +4.229, E3 +73977.760}
SPL {X  -159.990, Y  +379.485, Z    +0.000, E1    +0.028, E3 +73977.805}
SPL {X  -159.990, Y  +381.270, Z    +0.000, E1    -3.383, E3 +73977.822}
SPL {X  -159.990, Y  +384.811, Z    +0.000, E1   -11.531, E3 +73977.912}
SPL {X  -159.990, Y  +390.180, Z    +0.000, E1   -24.142, E3 +73978.216}
SPL {X  -159.990, Y  +397.074, Z    +0.000, E1   -39.012, E3 +73978.826}
SPL {X  -159.990, Y  +405.152, Z    +0.000, E1   -50.697, E3 +73979.965}
SPL {X  -159.990, Y  +423.293, Z    +0.000, E1   -63.280, E3 +73983.966}
SPL {X  -159.990, Y  +493.649, Z    +0.000, E1   -71.671, E3 +74009.670}
SPL {X  -159.990, Y  +662.531, Z    +0.000, E1   -73.010, E3 +74096.493}
SPL {X  -159.805, Y  +684.185, Z    +0.000, E1   -72.979, E3 +74110.777}
SPL {X  -158.295, Y  +699.729, Z    +0.000, E1   -72.830, E3 +74122.447}
SPL {X  -155.857, Y  +712.630, Z    +0.000, E1   -72.572, E3 +74133.376}
SPL {X  -153.206, Y  +722.596, Z    +0.000, E1   -72.287, E3 +74142.557}
SPL {X  -150.445, Y  +730.933, Z    +0.000, E1   -71.979, E3 +74150.768}
SPL {X  -147.389, Y  +738.737, Z    +0.000, E1   -71.634, E3 +74158.840}
SPL {X  -144.044, Y  +746.129, Z    +0.000, E1   -71.236, E3 +74166.835}
SPL {X  -140.684, Y  +752.689, Z    +0.000, E1   -70.820, E3 +74174.210}
SPL {X  -137.335, Y  +758.572, Z    +0.000, E1   -70.388, E3 +74181.017}
SPL {X  -133.651, Y  +764.444, Z    +0.000, E1   -69.897, E3 +74187.970}
SPL {X  -129.492, Y  +770.461, Z    +0.000, E1   -69.311, E3 +74195.210}
SPL {X  -125.168, Y  +776.148, Z    +0.000, E1   -68.666, E3 +74202.086}
SPL {X  -122.036, Y  +779.960, Z    +0.000, E1   -68.144, E3 +74206.689}
SPL {X   -80.879, Y  +814.541, Z    +0.000, E1   -55.704, E3 +74328.007}
ENDSPLINE

SPLINE
SPL {X  -125.518, Y  +775.707, Z    +0.000, E1   -52.189, E3 +74499.484}
SPL {X  -144.748, Y  +744.653, Z    +0.000, E1   -45.208, E3 +74517.680}
SPL {X  -153.147, Y  +722.791, Z    +0.000, E1   -36.417, E3 +74524.076}
SPL {X  -157.402, Y  +705.160, Z    +0.000, E1   -26.108, E3 +74527.171}
SPL {X  -159.480, Y  +689.270, Z    +0.000, E1   -14.023, E3 +74528.737}
SPL {X  -159.986, Y  +677.650, Z    +0.000, E1    -3.291, E3 +74529.231}
SPL {X  -159.990, Y  +674.500, Z    +0.000, E1    +0.000, E3 +74529.262}
SPL {X  -159.990, Y  +672.716, Z    +0.000, E1    +3.405, E3 +74529.278}
SPL {X  -159.990, Y  +668.521, Z    +0.000, E1   +13.007, E3 +74529.397}
SPL {X  -159.990, Y  +664.286, Z    +0.000, E1   +23.338, E3 +74529.629}
SPL {X  -159.990, Y  +658.431, Z    +0.000, E1   +35.998, E3 +74530.123}
SPL {X  -159.990, Y  +650.524, Z    +0.000, E1   +48.779, E3 +74531.112}
SPL {X  -159.990, Y  +641.022, Z    +0.000, E1   +57.726, E3 +74532.979}
SPL {X  -159.990, Y  +617.987, Z    +0.000, E1   +67.134, E3 +74538.874}
SPL {X  -159.990, Y  +532.407, Z    +0.000, E1   +73.084, E3 +74569.781}
SPL {X  -159.990, Y  +390.607, Z    +0.000, E1   +73.632, E3 +74641.317}
SPL {X  -159.886, Y  +371.742, Z    +0.000, E1   +73.650, E3 +74653.104}
SPL {X  -157.928, Y  +351.899, Z    +0.000, E1   +73.451, E3 +74667.537}
ENDSPLINE

SPLINE
SPL {X  -159.990, Y  +380.170, Z    +0.000, E1   +69.785, E3 +74683.678}
ENDSPLINE

SPLINE
SPL {X  -158.227, Y  +353.814, Z    +0.000, E1   +70.663, E3 +74695.571}
SPL {X  -154.257, Y  +335.055, Z    +0.000, E1   +71.089, E3 +74705.199}
SPL {X  -148.145, Y  +317.085, Z    +0.000, E1   +71.657, E3 +74712.369}
ENDSPLINE

SLIN {X  -200.000, Y  +530.000, E1    +0.000}
HALT
END
